"A_2111_KCL01_I2"	I 144.3	BOOL	// SCREW OFF
"A_2111_KCL01_I3"	I 144.4	BOOL	// DRIVE FORWARD SLOWLY
"A_2111_KCL01_I4"	I 144.5	BOOL	// DRIVE BACKWARD SLOWLY
"A_2115_KCL01_I1"	I 160.0	BOOL	// BACKWALL LIFTING
"A_2115_KCL01_I2"	I 160.1	BOOL	// BACKWALL LOWERING
"A_2115_KCL01_I3"	I 160.2	BOOL	// UNCOUPLE
"A_2115_KCL01_I4"	I 160.3	BOOL	// COUPLE
"A_2115_KCL01_I5"	I 160.4	BOOL	// WALL LOCKING
"A_2115_KCL01_I6"	I 160.5	BOOL	// WALL UNLOCKING
"A_2115_KCL01_I7"	I 160.6	BOOL	// HORIZONTAL SCREW ON
"A_2115_KCL01_I8"	I 160.7	BOOL	// DIAGONAL SCREW ON
"A_2115_KCL01_I9"	I 161.0	BOOL	// SCREW STOP
"A_2115_BSA12_I1"	I 161.2	BOOL	// ZERO SPEED MONITOR HORIZONTAL SCREW
"A_2115_BSA17_I1"	I 161.3	BOOL	// ZERO SPEED MONITOR LIFTING SCREW
"A_21_K838R1_I1"	I 162.0	BOOL	// FUSE SWITCH OFF +M212
"A_2199_SHE04_I1"	I 162.1	BOOL	// EMERGENCY-STOP 1 MACHINE DBFL
"A_2199_SHE05_I1"	I 162.2	BOOL	// EMERGENCY-STOP 2 MACHINE DBFL
"A_2199_SHE08_I1"	I 162.3	BOOL	// EMERGENCY-STOP 3 MACHINE DBFL
"A_2115_QYS18_I1"	I 162.4	BOOL	// CLEANING FLAP 1
"A_2115_QYS19_I1"	I 162.5	BOOL	// CLEANING FLAP 2
"A_2115_BTT11_I1"	I 162.6	BOOL	// THERMISTOR HORIZONTAL SCREW
"A_2115_BTT15_I1"	I 162.7	BOOL	// THERMISTOR LIFTING SCREW
"A_2115_BZS42_I1"	I 163.0	BOOL	// COUPLING DRIVE UNLOCKED
"A_2115_BZS43_I1"	I 163.1	BOOL	// COUPLING DRIVE LOCKED
"A_2115_BZS46_I1"	I 163.2	BOOL	// COUPLING DRIVE UNLOCKED
"A_2115_BZS47_I1"	I 163.3	BOOL	// COUPLING DRIVE LOCKED
"A_2150_MXZ01_I1"	I 164.0	BOOL	// AIR-FLAP 1 OPEN
"A_2150_MXZ01_I2"	I 164.1	BOOL	// AIR-FLAP 1 CLOSE
"A_2150_BZS01_I1"	I 164.2	BOOL	// AIR-FLAP 1 CLOSED
"A_2150_BZS02_I1"	I 164.3	BOOL	// AIR-FLAP 1 OPENED
"A_2151_MXZ01_I1"	I 164.4	BOOL	// AIR-FLAP 2 OPEN
"A_2151_MXZ01_I2"	I 164.5	BOOL	// AIR-FLAP 2 CLOSE
"A_2151_BZS01_I1"	I 164.6	BOOL	// AIR-FLAP 2 CLOSED
"A_2151_BZS02_I1"	I 164.7	BOOL	// AIR-FLAP 2 OPENED
"A_2152_MXZ01_I1"	I 165.0	BOOL	// AIR-FLAP 3 OPEN
"A_2152_MXZ01_I2"	I 165.1	BOOL	// AIR-FLAP 3 CLOSE
"A_2152_BZS01_I1"	I 165.2	BOOL	// AIR-FLAP 3 CLOSED
"A_2152_BZS02_I1"	I 165.3	BOOL	// AIR-FLAP 3 OPENED
"A_2154_MXZ01_I1"	I 165.4	BOOL	// WATER PUMP 1
"A_2155_MXZ01_I1"	I 165.5	BOOL	// WATER PUMP 2
"A_2160_MXZ01_I1"	I 165.6	BOOL	// GERM FAN 1
"A_2160_MXZ02_I1"	I 165.7	BOOL	// GERM FAN 2
"A_22_A040Z1_I1"	I 200.0	BOOL	// POWER SUPPLY FAILURE +C22
"A_22_S_H097Z1_I1"	I 200.1	BOOL	// OPERATING ON +C22
"A_22_K091Z1_I1"	I 200.2	BOOL	// FUSE SWITCH OFF +C22
"A_22_A097Z1_I1"	I 200.3	BOOL	// EMERGENCY-STOP +C22
"A_22_A098Z1_I1"	I 200.4	BOOL	// EMERGENCY-STOP +M221/M222
"A_22_Q390Z1_I1"	I 200.5	BOOL	// POWER SUPPLY MACHINE BMKE
"A_22_Q445Z1_I1"	I 200.6	BOOL	// POWER SUPPLY MACHINE DBFL
"A_22_D1B065_I1"	I 200.7	BOOL	// CONTROL 24VDC LIMIT SWITCHES WAY
"A_2299_SHE01_I1"	I 201.0	BOOL	// EMERGENCY-OFF CUSTOMER
"A_2299_SHE02_I1"	I 201.1	BOOL	// EMERGENCY-OFF CUSTOMER
"A_22_A700Z1_I1"	I 201.4	BOOL	// POWER CIRCUIT CABLE CHAIN
"A_22_A106Z1_I1"	I 201.5	BOOL	// EMERGENCY-STOP FROM +C21
"A_22_A800Z1_I1"	I 201.6	BOOL	// POWER CIRCUIT CABLE CHAIN
"A_2201_MXZ01_I1"	I 202.0	BOOL	// BELT CONVEYOR
"A_2202_YMXZ01_I1"	I 202.1	BOOL	// CHUTE DRIVE LEFT SIDE
"A_2202_YMXZ01_I2"	I 202.2	BOOL	// CHUTE DRIVE RIGHT SIDE
"A_2211_MXZ41_I1"	I 203.0	BOOL	// TRAVELING DRIVE
"A_2211_MXZ61_I1"	I 203.2	BOOL	// TURNING SCREW DRIVE 1
"A_2211_MXZ62_I1"	I 203.3	BOOL	// TURNING SCREW DRIVE 2
"A_2211_MXZ63_I1"	I 203.4	BOOL	// TURNING SCREW DRIVE 3
"A_2211_MXZ64_I1"	I 203.5	BOOL	// TURNING SCREW DRIVE 4
"A_2211_MXZ65_I1"	I 203.6	BOOL	// TURNING SCREW DRIVE 5
"A_2211_MXZ66_I1"	I 203.7	BOOL	// TURNING SCREW DRIVE 6
"A_2211_MXZ67_I1"	I 204.0	BOOL	// TURNING SCREW DRIVE 7
"A_2211_MXZ68_I1"	I 204.1	BOOL	// TURNING SCREW DRIVE 8
"A_2211_MXZ69_I1"	I 204.2	BOOL	// TURNING SCREW DRIVE 9
"A_2211_MXZ70_I1"	I 204.3	BOOL	// TURNING SCREW DRIVE 10
"A_2211_MXZ71_I1"	I 204.4	BOOL	// TURNING SCREW DRIVE 11
"A_2211_MXZ72_I1"	I 204.5	BOOL	// TURNING SCREW DRIVE 12
"A_2211_MXZ73_I1"	I 204.6	BOOL	// TURNING SCREW DRIVE 13
"A_2201_SHE20_I1"	I 205.0	BOOL	// CABLE PULL SWITCH RIGHT 1
"A_2201_SHE21_I1"	I 205.1	BOOL	// CABLE PULL SWITCH RIGHT 2
"A_2201_SHE22_I1"	I 205.2	BOOL	// CABLE PULL SWITCH LEFT 1
"A_2201_SHE23_I1"	I 205.3	BOOL	// CABLE PULL SWITCH LEFT 2
"A_2202_QYS21_I1"	I 205.5	BOOL	// DISCHARGE CHUTE LEFT SIDE
"A_2202_QYS22_I1"	I 205.6	BOOL	// DISCHARGE CHUTE RIGHT SIDE
"A_2215_MXZ11_I1"	I 208.0	BOOL	// HORIZONTAL SCREW
"A_2215_MXZ15_I1"	I 208.2	BOOL	// LIFTING SCREW
"A_2215_MXZ21_I1"	I 208.3	BOOL	// LIFTING DEVICE DOWN
"A_2215_MXZ21_I2"	I 208.4	BOOL	// LIFTING DEVICE UP
"A_22_A458Z1_I1"	I 210.0	BOOL	// CLEANING FLAP 1/2
"A_2215_BZS22_I1"	I 210.6	BOOL	// LIFTING DEVICE DOWN
"A_2215_BZS23_I1"	I 210.7	BOOL	// LIFTING DEVICE END POSITION TOP
"A_2245_QXV21_I1"	I 216.0	BOOL	// RUNNING COOLING UNIT GERMINATING
"A_2245_QXV31_I1"	I 216.1	BOOL	// RUNNING COOLING UNIT GERMINATING
"A_2216_BZS12_I1"	I 216.4	BOOL	// SPRINKING WATER LINE OPENED
"A_2216_BZS11_I1"	I 216.5	BOOL	// SPRINKING WATER LINE CLOSED
"A_2231_BZS12_I1"	I 217.2	BOOL	// VALVE HUMIDIFICATION OPENED
"A_2231_BZS11_I1"	I 217.3	BOOL	// VALVE HUMIDIFICATION CLOSED
"A_2201_BSA13_I1"	I 217.4	BOOL	// SPEED CONTROL
"A_2201_BZS14_15_I1"	I 217.6	BOOL	// BELT MONITOR RIGHT
"A_2201_BZS16_17_I1"	I 217.7	BOOL	// BELT MONITOR LEFT
"A_2202_BZS13_I1"	I 218.2	BOOL	// DISCHARGE CHUTE PARKING POSITION
"A_2202_BZS14_I1"	I 218.3	BOOL	// DISCHARGE CHUTE LEFT SIDE
"A_2202_BZS15_I1"	I 218.4	BOOL	// DISCHARGE CHUTE RIGHT SIDE
"A_2212_BZS12_I1"	I 240.0	BOOL	// SPRINKING WATER LINE 1 OPENED
"A_2212_BZS11_I1"	I 240.1	BOOL	// SPRINKING WATER LINE 1 CLOSED
"A_2212_BZS22_I1"	I 240.2	BOOL	// SPRINKING WATER LINE 2 OPENED
"A_2212_BZS21_I1"	I 240.3	BOOL	// SPRINKING WATER LINE 2 CLOSED
"A_2211_KCL01_I1"	I 240.4	BOOL	// SCREW ON
"A_2211_KCL01_I2"	I 240.5	BOOL	// SCREW OFF
"A_2211_KCL01_I3"	I 240.6	BOOL	// DRIVE FORWARD SLOWLY
"A_2211_KCL01_I4"	I 240.7	BOOL	// DRIVE BACKWARD SLOWLY
"A_2211_KCL01_I5"	I 241.0	BOOL	// DRIVE FORWARD FASTER
"A_2211_KCL01_I6"	I 241.1	BOOL	// DRIVE BACKWARD FASTER
"A_2211_BZS44_I1"	I 241.2	BOOL	// TRAVELING DRIVE STOP LEFT SIDE
"A_2211_BZS46_I1"	I 241.3	BOOL	// TRAVELING DRIVE STOP RIGHT SIDE
"A_22_K738R1_I1"	I 242.0	BOOL	// FUSE SWITCH OFF +M221
"A_22_A408Z1_I1"	I 242.1	BOOL	// BUMPER SWITCHED-OFF
"A_2299_SHE03_I1"	I 242.2	BOOL	// EMERGENCY-STOP 1 MACHINE BMKE
"A_2299_SHE06_I1"	I 242.3	BOOL	// EMERGENCY-STOP 2 MACHINE BMKE
"A_2211_QYS43_I1"	I 242.4	BOOL	// TRAVELING DRIVE SAFETY STLEFT SIDE
"A_2211_QYS45_I1"	I 242.5	BOOL	// TRAVELING DRIVE SAFETY STRIGHT SIDE
"A_2299_SHE20_I1"	I 242.6	BOOL	// CABLE PULL SWITCH RIGHT
"A_2299_SHE21_I1"	I 242.7	BOOL	// CABLE PULL SWITCH LEFT
"A_2211_BZS22_I1"	I 243.0	BOOL	// COUPLING DRIVE UNLOCKED
"A_2211_BZS23_I1"	I 243.1	BOOL	// COUPLING DRIVE LOCKED
"A_2211_BZS26_I1"	I 243.2	BOOL	// COUPLING DRIVE UNLOCKED
"A_2211_BZS27_I1"	I 243.3	BOOL	// COUPLING DRIVE LOCKED
"A_2211_BZS32_I1"	I 243.4	BOOL	// COUPLING DRIVE UNLOCKED
"A_2211_BZS33_I1"	I 243.5	BOOL	// COUPLING DRIVE LOCKED
"A_2211_BZS36_I1"	I 243.6	BOOL	// COUPLING DRIVE UNLOCKED
"A_2211_BZS37_I1"	I 243.7	BOOL	// COUPLING DRIVE LOCKED
"A_2215_KCL01_I1"	I 260.0	BOOL	// BACKWALL LIFTING
"A_2215_KCL01_I2"	I 260.1	BOOL	// BACKWALL LOWERING
"A_2215_KCL01_I3"	I 260.2	BOOL	// UNCOUPLE
"A_2215_KCL01_I4"	I 260.3	BOOL	// COUPLE
"A_2215_KCL01_I5"	I 260.4	BOOL	// WALL LOCKING
"A_2215_KCL01_I6"	I 260.5	BOOL	// WALL UNLOCKING
"A_2215_KCL01_I7"	I 260.6	BOOL	// HORIZONTAL SCREW ON
"A_2215_KCL01_I8"	I 260.7	BOOL	// DIAGONAL SCREW ON
"A_2215_KCL01_I9"	I 261.0	BOOL	// SCREW STOP
"A_2215_BSA12_I1"	I 261.2	BOOL	// ZERO SPEED MONITOR HORIZONTAL SCREW
"A_2215_BSA17_I1"	I 261.3	BOOL	// ZERO SPEED MONITOR LIFTING SCREW
"A_22_K838R1_I1"	I 262.0	BOOL	// FUSE SWITCH OFF +M222
"A_2299_SHE04_I1"	I 262.1	BOOL	// EMERGENCY-STOP 1 MACHINE DBFL
"A_2299_SHE05_I1"	I 262.2	BOOL	// EMERGENCY-STOP 2 MACHINE DBFL
"A_2299_SHE08_I1"	I 262.3	BOOL	// EMERGENCY-STOP 3 MACHINE DBFL
"A_2215_QYS18_I1"	I 262.4	BOOL	// CLEANING FLAP 1
"A_2215_QYS19_I1"	I 262.5	BOOL	// CLEANING FLAP 2
"A_2215_BTT11_I1"	I 262.6	BOOL	// THERMISTOR HORIZONTAL SCREW
"A_2215_BTT15_I1"	I 262.7	BOOL	// THERMISTOR LIFTING SCREW
"A_2215_BZS42_I1"	I 263.0	BOOL	// COUPLING DRIVE UNLOCKED
"A_2215_BZS43_I1"	I 263.1	BOOL	// COUPLING DRIVE LOCKED
"A_2215_BZS46_I1"	I 263.2	BOOL	// COUPLING DRIVE UNLOCKED
"A_2215_BZS47_I1"	I 263.3	BOOL	// COUPLING DRIVE LOCKED
"A_2250_MXZ01_I1"	I 264.0	BOOL	// AIR-FLAP 1 OPEN
"A_2250_MXZ01_I2"	I 264.1	BOOL	// AIR-FLAP 1 CLOSE
"A_2250_BZS01_I1"	I 264.2	BOOL	// AIR-FLAP 1 CLOSED
"A_2250_BZS02_I1"	I 264.3	BOOL	// AIR-FLAP 1 OPENED
"A_2251_MXZ01_I1"	I 264.4	BOOL	// AIR-FLAP 2 OPEN
"A_2251_MXZ01_I2"	I 264.5	BOOL	// AIR-FLAP 2 CLOSE
"A_2251_BZS01_I1"	I 264.6	BOOL	// AIR-FLAP 2 CLOSED
"A_2251_BZS02_I1"	I 264.7	BOOL	// AIR-FLAP 2 OPENED
"A_2252_MXZ01_I1"	I 265.0	BOOL	// AIR-FLAP 3 OPEN
"A_2252_MXZ01_I2"	I 265.1	BOOL	// AIR-FLAP 3 CLOSE
"A_2252_BZS01_I1"	I 265.2	BOOL	// AIR-FLAP 3 CLOSED
"A_2252_BZS02_I1"	I 265.3	BOOL	// AIR-FLAP 3 OPENED
"A_2254_MXZ01_I1"	I 265.4	BOOL	// WATER PUMP 1
"A_2255_MXZ01_I1"	I 265.5	BOOL	// WATER PUMP 2
"A_2260_MXZ01_I1"	I 265.6	BOOL	// GERM FAN 1
"A_2260_MXZ02_I1"	I 265.7	BOOL	// GERM FAN 2
"A_23_A040Z1_I1"	I 300.0	BOOL	// POWER SUPPLY FAILURE +C23
"A_23_S_H097Z1_I1"	I 300.1	BOOL	// OPERATING ON +C23
"A_23_K091Z1_I1"	I 300.2	BOOL	// FUSE SWITCH OFF +C23
"A_23_A097Z1_I1"	I 300.3	BOOL	// EMERGENCY-STOP +C23
"A_23_A098Z1_I1"	I 300.4	BOOL	// EMERGENCY-STOP +M231/M232
"A_23_Q390Z1_I1"	I 300.5	BOOL	// POWER SUPPLY MACHINE BMKE
"A_23_Q445Z1_I1"	I 300.6	BOOL	// POWER SUPPLY MACHINE DBFL
"A_23_D1B065_I1"	I 300.7	BOOL	// CONTROL 24VDC LIMIT SWITCHES WAY
"A_2399_SHE01_I1"	I 301.0	BOOL	// EMERGENCY-OFF CUSTOMER
"A_2399_SHE02_I1"	I 301.1	BOOL	// EMERGENCY-OFF CUSTOMER
"A_23_A700Z1_I1"	I 301.4	BOOL	// POWER CIRCUIT CABLE CHAIN
"A_23_A106Z1_I1"	I 301.5	BOOL	// EMERGENCY-STOP FROM +C24
"A_23_A800Z1_I1"	I 301.6	BOOL	// POWER CIRCUIT CABLE CHAIN
"A_2301_MXZ01_I1"	I 302.0	BOOL	// BELT CONVEYOR
"A_2302_YMXZ01_I1"	I 302.1	BOOL	// CHUTE DRIVE LEFT SIDE
"A_2302_YMXZ01_I2"	I 302.2	BOOL	// CHUTE DRIVE RIGHT SIDE
"A_2311_MXZ41_I1"	I 303.0	BOOL	// TRAVELING DRIVE
"A_2311_MXZ61_I1"	I 303.2	BOOL	// TURNING SCREW DRIVE 1
"A_2311_MXZ62_I1"	I 303.3	BOOL	// TURNING SCREW DRIVE 2
"A_2311_MXZ63_I1"	I 303.4	BOOL	// TURNING SCREW DRIVE 3
"A_2311_MXZ64_I1"	I 303.5	BOOL	// TURNING SCREW DRIVE 4
"A_2311_MXZ65_I1"	I 303.6	BOOL	// TURNING SCREW DRIVE 5
"A_2311_MXZ66_I1"	I 303.7	BOOL	// TURNING SCREW DRIVE 6
"A_2311_MXZ67_I1"	I 304.0	BOOL	// TURNING SCREW DRIVE 7
"A_2311_MXZ68_I1"	I 304.1	BOOL	// TURNING SCREW DRIVE 8
"A_2311_MXZ69_I1"	I 304.2	BOOL	// TURNING SCREW DRIVE 9
"A_2311_MXZ70_I1"	I 304.3	BOOL	// TURNING SCREW DRIVE 10
"A_2311_MXZ71_I1"	I 304.4	BOOL	// TURNING SCREW DRIVE 12
"A_2311_MXZ72_I1"	I 304.5	BOOL	// TURNING SCREW DRIVE 12
"A_2311_MXZ73_I1"	I 304.6	BOOL	// TURNING SCREW DRIVE 13
"A_2301_SHE20_I1"	I 305.0	BOOL	// CABLE PULL SWITCH RIGHT 1
"A_2301_SHE21_I1"	I 305.1	BOOL	// CABLE PULL SWITCH RIGHT 2
"A_2301_SHE22_I1"	I 305.2	BOOL	// CABLE PULL SWITCH LEFT 1
"A_2301_SHE23_I1"	I 305.3	BOOL	// CABLE PULL SWITCH LEFT 2
"A_2302_QYS21_I1"	I 305.5	BOOL	// DISCHARGE CHUTE LEFT SIDE
"A_2302_QYS22_I1"	I 305.6	BOOL	// DISCHARGE CHUTE RIGHT SIDE
"A_2315_MXZ11_I1"	I 308.0	BOOL	// HORIZONTAL SCREW
"A_2315_MXZ15_I1"	I 308.2	BOOL	// LIFTING SCREW
"A_2315_MXZ21_I1"	I 308.3	BOOL	// LIFTING DEVICE DOWN
"A_2315_MXZ21_I2"	I 308.4	BOOL	// LIFTING DEVICE UP
"A_23_A458Z1_I1"	I 310.0	BOOL	// CLEANING FLAP 1/2
"A_2315_BZS22_I1"	I 310.6	BOOL	// LIFTING DEVICE DOWN
"A_2315_BZS23_I1"	I 310.7	BOOL	// LIFTING DEVICE END POSITION TOP
"A_2345_QXV21_I1"	I 316.0	BOOL	// RUNNING COOLING UNIT GERMINATING
"A_2345_QXV31_I1"	I 316.1	BOOL	// RUNNING COOLING UNIT GERMINATING
"A_2316_BZS12_I1"	I 316.4	BOOL	// SPRINKING WATER LINE OPENED
"A_2316_BZS11_I1"	I 316.5	BOOL	// SPRINKING WATER LINE CLOSED
"A_2331_BZS12_I1"	I 317.2	BOOL	// VALVE HUMIDIFICATION OPENED
"A_2331_BZS11_I1"	I 317.3	BOOL	// VALVE HUMIDIFICATION CLOSED
"A_2301_BSA13_I1"	I 317.4	BOOL	// SPEED CONTROL
"A_2301_BZS14_15_I1"	I 317.6	BOOL	// BELT MONITOR RIGHT
"A_2301_BZS16_17_I1"	I 317.7	BOOL	// BELT MONITOR LEFT
"A_2302_BZS13_I1"	I 318.2	BOOL	// DISCHARGE CHUTE PARKING POSITION
"A_2302_BZS14_I1"	I 318.3	BOOL	// DISCHARGE CHUTE LEFT SIDE
"A_2302_BZS15_I1"	I 318.4	BOOL	// DISCHARGE CHUTE RIGHT SIDE
"A_2312_BZS12_I1"	I 340.0	BOOL	// SPRINKING WATER LINE 1 OPENED
"A_2312_BZS11_I1"	I 340.1	BOOL	// SPRINKING WATER LINE 1 CLOSED
"A_2312_BZS22_I1"	I 340.2	BOOL	// SPRINKING WATER LINE 2 OPENED
"A_2312_BZS21_I1"	I 340.3	BOOL	// SPRINKING WATER LINE 2 CLOSED
"A_2311_KCL01_I1"	I 340.4	BOOL	// SCREW ON
"A_2311_KCL01_I2"	I 340.5	BOOL	// SCREW OFF
"A_2311_KCL01_I3"	I 340.6	BOOL	// DRIVE FORWARD SLOWLY
"A_2311_KCL01_I4"	I 340.7	BOOL	// DRIVE BACKWARD SLOWLY
"A_2311_KCL01_I5"	I 341.0	BOOL	// DRIVE FORWARD FASTER
"A_2311_KCL01_I6"	I 341.1	BOOL	// DRIVE BACKWARD FASTER
"A_2311_BZS44_I1"	I 341.2	BOOL	// TRAVELING DRIVE STOP LEFT SIDE
"A_2311_BZS46_I1"	I 341.3	BOOL	// TRAVELING DRIVE STOP RIGHT SIDE
"A_23_K738R1_I1"	I 342.0	BOOL	// FUSE SWITCH OFF +M231
"A_23_A408Z1_I1"	I 342.1	BOOL	// BUMPER SWITCHED-OFF
"A_2399_SHE03_I1"	I 342.2	BOOL	// EMERGENCY-STOP 1 MACHINE BMKE
"A_2399_SHE06_I1"	I 342.3	BOOL	// EMERGENCY-STOP 2 MACHINE BMKE
"A_2311_QYS43_I1"	I 342.4	BOOL	// TRAVELING DRIVE SAFETY STLEFT SIDE
"A_2311_QYS45_I1"	I 342.5	BOOL	// TRAVELING DRIVE SAFETY STRIGHT SIDE
"A_2399_SHE20_I1"	I 342.6	BOOL	// CABLE PULL SWITCH RIGHT
"A_2399_SHE21_I1"	I 342.7	BOOL	// CABLE PULL SWITCH LEFT
"A_2311_BZS22_I1"	I 343.0	BOOL	// COUPLING DRIVE UNLOCKED
"A_2311_BZS23_I1"	I 343.1	BOOL	// COUPLING DRIVE LOCKED
"A_2311_BZS26_I1"	I 343.2	BOOL	// COUPLING DRIVE UNLOCKED
"A_2311_BZS27_I1"	I 343.3	BOOL	// COUPLING DRIVE LOCKED
"A_2311_BZS32_I1"	I 343.4	BOOL	// COUPLING DRIVE UNLOCKED
"A_2311_BZS33_I1"	I 343.5	BOOL	// COUPLING DRIVE LOCKED
"A_2311_BZS36_I1"	I 343.6	BOOL	// COUPLING DRIVE UNLOCKED
"A_2311_BZS37_I1"	I 343.7	BOOL	// COUPLING DRIVE LOCKED
"A_2315_KCL01_I1"	I 360.0	BOOL	// BACKWALL LIFTING
"A_2315_KCL01_I2"	I 360.1	BOOL	// BACKWALL LOWERING
"A_2315_KCL01_I3"	I 360.2	BOOL	// UNCOUPLE
"A_2315_KCL01_I4"	I 360.3	BOOL	// COUPLE
"A_2315_KCL01_I5"	I 360.4	BOOL	// WALL LOCKING
"A_2315_KCL01_I6"	I 360.5	BOOL	// WALL UNLOCKING
"A_2315_KCL01_I7"	I 360.6	BOOL	// HORIZONTAL SCREW ON
"A_2315_KCL01_I8"	I 360.7	BOOL	// DIAGONAL SCREW ON
"A_2315_KCL01_I9"	I 361.0	BOOL	// SCREW STOP
"A_2315_BSA12_I1"	I 361.2	BOOL	// ZERO SPEED MONITOR HORIZONTAL SCREW
"A_2315_BSA17_I1"	I 361.3	BOOL	// ZERO SPEED MONITOR LIFTING SCREW
"A_23_K838R1_I1"	I 362.0	BOOL	// FUSE SWITCH OFF +M232
"A_2399_SHE04_I1"	I 362.1	BOOL	// EMERGENCY-STOP 1 MACHINE DBFL
"A_2399_SHE05_I1"	I 362.2	BOOL	// EMERGENCY-STOP 2 MACHINE DBFL
"A_2399_SHE08_I1"	I 362.3	BOOL	// EMERGENCY-STOP 3 MACHINE DBFL
"A_2315_QYS18_I1"	I 362.4	BOOL	// CLEANING FLAP 1
"A_2315_QYS19_I1"	I 362.5	BOOL	// CLEANING FLAP 2
"A_2315_BTT11_I1"	I 362.6	BOOL	// THERMISTOR HORIZONTAL SCREW
"A_2315_BTT15_I1"	I 362.7	BOOL	// THERMISTOR LIFTING SCREW
"A_2315_BZS42_I1"	I 363.0	BOOL	// COUPLING DRIVE UNLOCKED
"A_2315_BZS43_I1"	I 363.1	BOOL	// COUPLING DRIVE LOCKED
"A_2315_BZS46_I1"	I 363.2	BOOL	// COUPLING DRIVE UNLOCKED
"A_2315_BZS47_I1"	I 363.3	BOOL	// COUPLING DRIVE LOCKED
"A_2350_MXZ01_I1"	I 364.0	BOOL	// AIR-FLAP 1 OPEN
"A_2350_MXZ01_I2"	I 364.1	BOOL	// AIR-FLAP 1 CLOSE
"A_2350_BZS01_I1"	I 364.2	BOOL	// AIR-FLAP 1 CLOSED
"A_2350_BZS02_I1"	I 364.3	BOOL	// AIR-FLAP 1 OPENED
"A_2351_MXZ01_I1"	I 364.4	BOOL	// AIR-FLAP 2 OPEN
"A_2351_MXZ01_I2"	I 364.5	BOOL	// AIR-FLAP 2 CLOSE
"A_2351_BZS01_I1"	I 364.6	BOOL	// AIR-FLAP 2 CLOSED
"A_2351_BZS02_I1"	I 364.7	BOOL	// AIR-FLAP 2 OPENED
"A_2352_MXZ01_I1"	I 365.0	BOOL	// AIR-FLAP 3 OPEN
"A_2352_MXZ01_I2"	I 365.1	BOOL	// AIR-FLAP 3 CLOSE
"A_2352_BZS01_I1"	I 365.2	BOOL	// AIR-FLAP 3 CLOSED
"A_2352_BZS02_I1"	I 365.3	BOOL	// AIR-FLAP 3 OPENED
"A_2354_MXZ01_I1"	I 365.4	BOOL	// WATER PUMP 1
"A_2355_MXZ01_I1"	I 365.5	BOOL	// WATER PUMP 2
"A_2360_MXZ01_I1"	I 365.6	BOOL	// GERM FAN 1
"A_2360_MXZ02_I1"	I 365.7	BOOL	// GERM FAN 2
"A_24_A040Z1_I1"	I 400.0	BOOL	// POWER SUPPLY FAILURE +C24
"A_24_S_H097Z1_I1"	I 400.1	BOOL	// OPERATING ON +C24
"A_24_K091Z1_I1"	I 400.2	BOOL	// FUSE SWITCH OFF +C24
"A_24_A097Z1_I1"	I 400.3	BOOL	// EMERGENCY-STOP +C24
"A_24_A098Z1_I1"	I 400.4	BOOL	// EMERGENCY-STOP +M241/M242
"A_24_Q390Z1_I1"	I 400.5	BOOL	// POWER SUPPLY MACHINE BMKE
"A_24_Q445Z1_I1"	I 400.6	BOOL	// POWER SUPPLY MACHINE DBFL
"A_24_D1B065_I1"	I 400.7	BOOL	// CONTROL 24VDC LIMIT SWITCHES WAY
"A_2499_SHE01_I1"	I 401.0	BOOL	// EMERGENCY-OFF CUSTOMER
"A_2499_SHE02_I1"	I 401.1	BOOL	// EMERGENCY-OFF CUSTOMER
"A_24_A700Z1_I1"	I 401.4	BOOL	// POWER CIRCUIT CABLE CHAIN
"A_24_A106Z1_I1"	I 401.5	BOOL	// EMERGENCY-STOP FROM +C23
"A_24_A800Z1_I1"	I 401.6	BOOL	// POWER CIRCUIT CABLE CHAIN
"A_2401_MXZ01_I1"	I 402.0	BOOL	// BELT CONVEYOR
"A_2402_YMXZ01_I1"	I 402.1	BOOL	// CHUTE DRIVE LEFT SIDE
"A_2402_YMXZ01_I2"	I 402.2	BOOL	// CHUTE DRIVE RIGHT SIDE
"A_2411_MXZ41_I1"	I 403.0	BOOL	// TRAVELING DRIVE
"A_2411_MXZ61_I1"	I 403.2	BOOL	// TURNING SCREW DRIVE 1
"A_2411_MXZ62_I1"	I 403.3	BOOL	// TURNING SCREW DRIVE 2
"A_2411_MXZ63_I1"	I 403.4	BOOL	// TURNING SCREW DRIVE 3
"A_2411_MXZ64_I1"	I 403.5	BOOL	// TURNING SCREW DRIVE 4
"A_2411_MXZ65_I1"	I 403.6	BOOL	// TURNING SCREW DRIVE 5
"A_2411_MXZ66_I1"	I 403.7	BOOL	// TURNING SCREW DRIVE 6
"A_2411_MXZ67_I1"	I 404.0	BOOL	// TURNING SCREW DRIVE 7
"A_2411_MXZ68_I1"	I 404.1	BOOL	// TURNING SCREW DRIVE 8
"A_2411_MXZ69_I1"	I 404.2	BOOL	// TURNING SCREW DRIVE 9
"A_2411_MXZ70_I1"	I 404.3	BOOL	// TURNING SCREW DRIVE 10
"A_2411_MXZ71_I1"	I 404.4	BOOL	// TURNING SCREW DRIVE 11
"A_2411_MXZ72_I1"	I 404.5	BOOL	// TURNING SCREW DRIVE 12
"A_2411_MXZ73_I1"	I 404.6	BOOL	// TURNING SCREW DRIVE 13
"A_2401_SHE20_I1"	I 405.0	BOOL	// CABLE PULL SWITCH RIGHT 1
"A_2401_SHE21_I1"	I 405.1	BOOL	// CABLE PULL SWITCH RIGHT 2
"A_2401_SHE22_I1"	I 405.2	BOOL	// CABLE PULL SWITCH LEFT 1
"A_2401_SHE23_I1"	I 405.3	BOOL	// CABLE PULL SWITCH LEFT 2
"A_2402_QYS21_I1"	I 405.5	BOOL	// DISCHARGE CHUTE LEFT SIDE
"A_2402_QYS22_I1"	I 405.6	BOOL	// DISCHARGE CHUTE RIGHT SIDE
"A_2415_MXZ11_I1"	I 408.0	BOOL	// HORIZONTAL SCREW
"A_2415_MXZ15_I1"	I 408.2	BOOL	// LIFTING SCREW
"A_2415_MXZ21_I1"	I 408.3	BOOL	// LIFTING DEVICE DOWN
"A_2415_MXZ21_I2"	I 408.4	BOOL	// LIFTING DEVICE UP
"A_24_A458Z1_I1"	I 410.0	BOOL	// CLEANING FLAP 1/2
"A_2415_BZS22_I1"	I 410.6	BOOL	// LIFTING DEVICE DOWN
"A_2415_BZS23_I1"	I 410.7	BOOL	// LIFTING DEVICE END POSITION TOP
"A_2445_QXV21_I1"	I 416.0	BOOL	// RUNNING COOLING UNIT GERMINATING
"A_2445_QXV31_I1"	I 416.1	BOOL	// RUNNING COOLING UNIT GERMINATING
"A_2416_BZS12_I1"	I 416.4	BOOL	// SPRINKING WATER LINE OPENED
"A_2416_BZS11_I1"	I 416.5	BOOL	// SPRINKING WATER LINE CLOSED
"A_2431_BZS12_I1"	I 417.2	BOOL	// VALVE HUMIDIFICATION OPENED
"A_2431_BZS11_I1"	I 417.3	BOOL	// VALVE HUMIDIFICATION CLOSED
"A_2401_BSA13_I1"	I 417.4	BOOL	// SPEED CONTROL
"A_2401_BZS14_15_I1"	I 417.6	BOOL	// BELT MONITOR RIGHT
"A_2401_BZS16_17_I1"	I 417.7	BOOL	// BELT MONITOR LEFT
"A_2402_BZS13_I1"	I 418.2	BOOL	// DISCHARGE CHUTE PARKING POSITION
"A_2402_BZS14_I1"	I 418.3	BOOL	// DISCHARGE CHUTE LEFT SIDE
"A_2402_BZS15_I1"	I 418.4	BOOL	// DISCHARGE CHUTE RIGHT SIDE
"A_2412_BZS12_I1"	I 440.0	BOOL	// SPRINKING WATER LINE 1 OPENED
"A_2412_BZS11_I1"	I 440.1	BOOL	// SPRINKING WATER LINE 1 CLOSED
"A_2412_BZS22_I1"	I 440.2	BOOL	// SPRINKING WATER LINE 2 OPENED
"A_2412_BZS21_I1"	I 440.3	BOOL	// SPRINKING WATER LINE 2 CLOSED
"A_2411_KCL01_I1"	I 440.4	BOOL	// SCREW ON
"A_2411_KCL01_I2"	I 440.5	BOOL	// SCREW OFF
"A_2411_KCL01_I3"	I 440.6	BOOL	// DRIVE FORWARD SLOWLY
"A_2411_KCL01_I4"	I 440.7	BOOL	// DRIVE BACKWARD SLOWLY
"A_2411_KCL01_I5"	I 441.0	BOOL	// DRIVE FORWARD FASTER
"A_2411_KCL01_I6"	I 441.1	BOOL	// DRIVE BACKWARD FASTER
"A_2411_BZS44_I1"	I 441.2	BOOL	// TRAVELING DRIVE STOP LEFT SIDE
"A_2411_BZS46_I1"	I 441.3	BOOL	// TRAVELING DRIVE STOP RIGHT SIDE
"A_24_K738R1_I1"	I 442.0	BOOL	// FUSE SWITCH OFF +M241
"A_24_A408Z1_I1"	I 442.1	BOOL	// BUMPER SWITCHED-OFF
"A_2499_SHE03_I1"	I 442.2	BOOL	// EMERGENCY-STOP 1 MACHINE BMKE
"A_2499_SHE06_I1"	I 442.3	BOOL	// EMERGENCY-STOP 2 MACHINE BMKE
"A_2411_QYS43_I1"	I 442.4	BOOL	// TRAVELING DRIVE SAFETY STLEFT SIDE
"A_2411_QYS45_I1"	I 442.5	BOOL	// TRAVELING DRIVE SAFETY STRIGHT SIDE
"A_2499_SHE20_I1"	I 442.6	BOOL	// CABLE PULL SWITCH RIGHT
"A_2499_SHE21_I1"	I 442.7	BOOL	// CABLE PULL SWITCH LEFT
"A_2411_BZS22_I1"	I 443.0	BOOL	// COUPLING DRIVE UNLOCKED
"A_2411_BZS23_I1"	I 443.1	BOOL	// COUPLING DRIVE LOCKED
"A_2411_BZS26_I1"	I 443.2	BOOL	// COUPLING DRIVE UNLOCKED
"A_2411_BZS27_I1"	I 443.3	BOOL	// COUPLING DRIVE LOCKED
"A_2411_BZS32_I1"	I 443.4	BOOL	// COUPLING DRIVE UNLOCKED
"A_2411_BZS33_I1"	I 443.5	BOOL	// COUPLING DRIVE LOCKED
"A_2411_BZS36_I1"	I 443.6	BOOL	// COUPLING DRIVE UNLOCKED
"A_2411_BZS37_I1"	I 443.7	BOOL	// COUPLING DRIVE LOCKED
"A_2415_KCL01_I1"	I 460.0	BOOL	// BACKWALL LIFTING
"A_2415_KCL01_I2"	I 460.1	BOOL	// BACKWALL LOWERING
"A_2415_KCL01_I3"	I 460.2	BOOL	// UNCOUPLE
"A_2415_KCL01_I4"	I 460.3	BOOL	// COUPLE
"A_2415_KCL01_I5"	I 460.4	BOOL	// WALL LOCKING
"A_2415_KCL01_I6"	I 460.5	BOOL	// WALL UNLOCKING
"A_2415_KCL01_I7"	I 460.6	BOOL	// HORIZONTAL SCREW ON
"A_2415_KCL01_I8"	I 460.7	BOOL	// DIAGONAL SCREW ON
"A_2415_KCL01_I9"	I 461.0	BOOL	// SCREW STOP
"A_2415_BSA12_I1"	I 461.2	BOOL	// ZERO SPEED MONITOR HORIZONTAL SCREW
"A_2415_BSA17_I1"	I 461.3	BOOL	// ZERO SPEED MONITOR LIFTING SCREW
"A_24_K838R1_I1"	I 462.0	BOOL	// FUSE SWITCH OFF +M242
"A_2499_SHE04_I1"	I 462.1	BOOL	// EMERGENCY-STOP 1 MACHINE DBFL
"A_2499_SHE05_I1"	I 462.2	BOOL	// EMERGENCY-STOP 2 MACHINE DBFL
"A_2499_SHE08_I1"	I 462.3	BOOL	// EMERGENCY-STOP 3 MACHINE DBFL
"A_2415_QYS18_I1"	I 462.4	BOOL	// CLEANING FLAP 1
"A_2415_QYS19_I1"	I 462.5	BOOL	// CLEANING FLAP 2
"A_2415_BTT11_I1"	I 462.6	BOOL	// THERMISTOR HORIZONTAL SCREW
"A_2415_BTT15_I1"	I 462.7	BOOL	// THERMISTOR LIFTING SCREW
"A_2415_BZS42_I1"	I 463.0	BOOL	// COUPLING DRIVE UNLOCKED
"A_2415_BZS43_I1"	I 463.1	BOOL	// COUPLING DRIVE LOCKED
"A_2415_BZS46_I1"	I 463.2	BOOL	// COUPLING DRIVE UNLOCKED
"A_2415_BZS47_I1"	I 463.3	BOOL	// COUPLING DRIVE LOCKED
"A_2450_MXZ01_I1"	I 464.0	BOOL	// AIR-FLAP 1 OPEN
"A_2450_MXZ01_I2"	I 464.1	BOOL	// AIR-FLAP 1 CLOSE
"A_2450_BZS01_I1"	I 464.2	BOOL	// AIR-FLAP 1 CLOSED
"A_2450_BZS02_I1"	I 464.3	BOOL	// AIR-FLAP 1 OPENED
"A_2451_MXZ01_I1"	I 464.4	BOOL	// AIR-FLAP 2 OPEN
"A_2451_MXZ01_I2"	I 464.5	BOOL	// AIR-FLAP 2 CLOSE
"A_2451_BZS01_I1"	I 464.6	BOOL	// AIR-FLAP 2 CLOSED
"A_2451_BZS02_I1"	I 464.7	BOOL	// AIR-FLAP 2 OPENED
"A_2452_MXZ01_I1"	I 465.0	BOOL	// AIR-FLAP 3 OPEN
"A_2452_MXZ01_I2"	I 465.1	BOOL	// AIR-FLAP 3 CLOSE
"A_2452_BZS01_I1"	I 465.2	BOOL	// AIR-FLAP 3 CLOSED
"A_2452_BZS02_I1"	I 465.3	BOOL	// AIR-FLAP 3 OPENED
"A_2454_MXZ01_I1"	I 465.4	BOOL	// WATER PUMP 1
"A_2455_MXZ01_I1"	I 465.5	BOOL	// WATER PUMP 2
"A_2460_MXZ01_I1"	I 465.6	BOOL	// GERM FAN 1
"A_2460_MXZ02_I1"	I 465.7	BOOL	// GERM FAN 2
"A_25_A040Z1_I1"	I 500.0	BOOL	// POWER SUPPLY FAILURE +C25
"A_25_S_H097Z1_I1"	I 500.1	BOOL	// OPERATING ON +C25
"A_25_K091Z1_I1"	I 500.2	BOOL	// FUSE SWITCH OFF +C25
"A_25_A097Z1_I1"	I 500.3	BOOL	// EMERGENCY-STOP +C25
"A_25_A098Z1_I1"	I 500.4	BOOL	// EMERGENCY-STOP +M251/M252
"A_25_Q390Z1_I1"	I 500.5	BOOL	// POWER SUPPLY MACHINE BMKE
"A_25_Q445Z1_I1"	I 500.6	BOOL	// POWER SUPPLY MACHINE DBFL
"A_25_D1B065_I1"	I 500.7	BOOL	// CONTROL 24VDC LIMIT SWITCHES WAY
"A_2599_SHE01_I1"	I 501.0	BOOL	// EMERGENCY-OFF CUSTOMER
"A_2599_SHE02_I1"	I 501.1	BOOL	// EMERGENCY-OFF CUSTOMER
"A_25_A700Z1_I1"	I 501.4	BOOL	// POWER CIRCUIT CABLE CHAIN
"A_25_A106Z1_I1"	I 501.5	BOOL	// EMERGENCY-STOP FROM +C26
"A_25_A800Z1_I1"	I 501.6	BOOL	// POWER CIRCUIT CABLE CHAIN
"A_2501_MXZ01_I1"	I 502.0	BOOL	// BELT CONVEYOR
"A_2502_YMXZ01_I1"	I 502.1	BOOL	// CHUTE DRIVE LEFT SIDE
"A_2502_YMXZ01_I2"	I 502.2	BOOL	// CHUTE DRIVE RIGHT SIDE
"A_2511_MXZ41_I1"	I 503.0	BOOL	// TRAVELING DRIVE
"A_2511_MXZ61_I1"	I 503.2	BOOL	// TURNING SCREW DRIVE 1
"A_2511_MXZ62_I1"	I 503.3	BOOL	// TURNING SCREW DRIVE 2
"A_2511_MXZ63_I1"	I 503.4	BOOL	// TURNING SCREW DRIVE 3
"A_2511_MXZ64_I1"	I 503.5	BOOL	// TURNING SCREW DRIVE 4
"A_2511_MXZ65_I1"	I 503.6	BOOL	// TURNING SCREW DRIVE 5
"A_2511_MXZ66_I1"	I 503.7	BOOL	// TURNING SCREW DRIVE 6
"A_2511_MXZ67_I1"	I 504.0	BOOL	// TURNING SCREW DRIVE 7
"A_2511_MXZ68_I1"	I 504.1	BOOL	// TURNING SCREW DRIVE 8
"A_2511_MXZ69_I1"	I 504.2	BOOL	// TURNING SCREW DRIVE 9
"A_2511_MXZ70_I1"	I 504.3	BOOL	// TURNING SCREW DRIVE 10
"A_2511_MXZ71_I1"	I 504.4	BOOL	// TURNING SCREW DRIVE 11
"A_2511_MXZ72_I1"	I 504.5	BOOL	// TURNING SCREW DRIVE 12
"A_2511_MXZ73_I1"	I 504.6	BOOL	// TURNING SCREW DRIVE 13
"A_2501_SHE20_I1"	I 505.0	BOOL	// CABLE PULL SWITCH RIGHT 1
"A_2501_SHE21_I1"	I 505.1	BOOL	// CABLE PULL SWITCH RIGHT 2
"A_2501_SHE22_I1"	I 505.2	BOOL	// CABLE PULL SWITCH LEFT 1
"A_2501_SHE23_I1"	I 505.3	BOOL	// CABLE PULL SWITCH LEFT 2
"A_2502_QYS21_I1"	I 505.5	BOOL	// DISCHARGE CHUTE LEFT SIDE
"A_2502_QYS22_I1"	I 505.6	BOOL	// DISCHARGE CHUTE RIGHT SIDE
"A_2515_MXZ11_I1"	I 508.0	BOOL	// HORIZONTAL SCREW
"A_2515_MXZ15_I1"	I 508.2	BOOL	// LIFTING SCREW
"A_2515_MXZ21_I1"	I 508.3	BOOL	// LIFTING DEVICE DOWN
"A_2515_MXZ21_I2"	I 508.4	BOOL	// LIFTING DEVICE UP
"A_25_A458Z1_I1"	I 510.0	BOOL	// CLEANING FLAP 1/2
"A_2515_BZS22_I1"	I 510.6	BOOL	// LIFTING DEVICE DOWN
"A_2515_BZS23_I1"	I 510.7	BOOL	// LIFTING DEVICE END POSITION TOP
"A_2545_QXV21_I1"	I 516.0	BOOL	// RUNNING COOLING UNIT GERMINATING
"A_2545_QXV31_I1"	I 516.1	BOOL	// RUNNING COOLING UNIT GERMINATING
"A_2516_BZS12_I1"	I 516.4	BOOL	// SPRINKING WATER LINE OPENED
"A_2516_BZS11_I1"	I 516.5	BOOL	// SPRINKING WATER LINE CLOSED
"A_2531_BZS12_I1"	I 517.2	BOOL	// VALVE HUMIDIFICATION OPENED
"A_2531_BZS11_I1"	I 517.3	BOOL	// VALVE HUMIDIFICATION CLOSED
"A_2501_BSA13_I1"	I 517.4	BOOL	// SPEED CONTROL
"A_2501_BZS14_15_I1"	I 517.6	BOOL	// BELT MONITOR RIGHT
"A_2501_BZS16_17_I1"	I 517.7	BOOL	// BELT MONITOR LEFT
"A_2502_BZS13_I1"	I 518.2	BOOL	// DISCHARGE CHUTE PARKING POSITION
"A_2502_BZS14_I1"	I 518.3	BOOL	// DISCHARGE CHUTE LEFT SIDE
"A_2502_BZS15_I1"	I 518.4	BOOL	// DISCHARGE CHUTE RIGHT SIDE
"A_2512_BZS12_I1"	I 540.0	BOOL	// SPRINKING WATER LINE 1 OPENED
"A_2512_BZS11_I1"	I 540.1	BOOL	// SPRINKING WATER LINE 1 CLOSED
"A_2512_BZS22_I1"	I 540.2	BOOL	// SPRINKING WATER LINE 2 OPENED
"A_2512_BZS21_I1"	I 540.3	BOOL	// SPRINKING WATER LINE 2 CLOSED
"A_2511_KCL01_I1"	I 540.4	BOOL	// SCREW ON
"A_2511_KCL01_I2"	I 540.5	BOOL	// SCREW OFF
"A_2511_KCL01_I3"	I 540.6	BOOL	// DRIVE FORWARD SLOWLY
"A_2511_KCL01_I4"	I 540.7	BOOL	// DRIVE BACKWARD SLOWLY
"A_2511_KCL01_I5"	I 541.0	BOOL	// DRIVE FORWARD FASTER
"A_2511_KCL01_I6"	I 541.1	BOOL	// DRIVE BACKWARD FASTER
"A_2511_BZS44_I1"	I 541.2	BOOL	// TRAVELING DRIVE STOP LEFT SIDE
"A_2511_BZS46_I1"	I 541.3	BOOL	// TRAVELING DRIVE STOP RIGHT SIDE
"A_25_K738R1_I1"	I 542.0	BOOL	// FUSE SWITCH OFF +M251
"A_25_A408Z1_I1"	I 542.1	BOOL	// BUMPER SWITCHED-OFF
"A_2599_SHE03_I1"	I 542.2	BOOL	// EMERGENCY-STOP 1 MACHINE BMKE
"A_2599_SHE06_I1"	I 542.3	BOOL	// EMERGENCY-STOP 2 MACHINE BMKE
"A_2511_QYS43_I1"	I 542.4	BOOL	// TRAVELING DRIVE SAFETY STLEFT SIDE
"A_2511_QYS45_I1"	I 542.5	BOOL	// TRAVELING DRIVE SAFETY STRIGHT SIDE
"A_2599_SHE20_I1"	I 542.6	BOOL	// CABLE PULL SWITCH RIGHT
"A_2599_SHE21_I1"	I 542.7	BOOL	// CABLE PULL SWITCH LEFT
"A_2511_BZS22_I1"	I 543.0	BOOL	// COUPLING DRIVE UNLOCKED
"A_2511_BZS23_I1"	I 543.1	BOOL	// COUPLING DRIVE LOCKED
"A_2511_BZS26_I1"	I 543.2	BOOL	// COUPLING DRIVE UNLOCKED
"A_2511_BZS27_I1"	I 543.3	BOOL	// COUPLING DRIVE LOCKED
"A_2511_BZS32_I1"	I 543.4	BOOL	// COUPLING DRIVE UNLOCKED
"A_2511_BZS33_I1"	I 543.5	BOOL	// COUPLING DRIVE LOCKED
"A_2511_BZS36_I1"	I 543.6	BOOL	// COUPLING DRIVE UNLOCKED
"A_2511_BZS37_I1"	I 543.7	BOOL	// COUPLING DRIVE LOCKED
"A_2515_KCL01_I1"	I 560.0	BOOL	// BACKWALL LIFTING
"A_2515_KCL01_I2"	I 560.1	BOOL	// BACKWALL LOWERING
"A_2515_KCL01_I3"	I 560.2	BOOL	// UNCOUPLE
"A_2515_KCL01_I4"	I 560.3	BOOL	// COUPLE
"A_2515_KCL01_I5"	I 560.4	BOOL	// WALL LOCKING
"A_2515_KCL01_I6"	I 560.5	BOOL	// WALL UNLOCKING
"A_2515_KCL01_I7"	I 560.6	BOOL	// HORIZONTAL SCREW ON
"A_2515_KCL01_I8"	I 560.7	BOOL	// DIAGONAL SCREW ON
"A_2515_KCL01_I9"	I 561.0	BOOL	// SCREW STOP
"A_2515_BSA12_I1"	I 561.2	BOOL	// ZERO SPEED MONITOR HORIZONTAL SCREW
"A_2515_BSA17_I1"	I 561.3	BOOL	// ZERO SPEED MONITOR LIFTING SCREW
"A_25_K838R1_I1"	I 562.0	BOOL	// FUSE SWITCH OFF +M252
"A_2599_SHE04_I1"	I 562.1	BOOL	// EMERGENCY-STOP 1 MACHINE DBFL
"A_2599_SHE05_I1"	I 562.2	BOOL	// EMERGENCY-STOP 2 MACHINE DBFL
"A_2599_SHE08_I1"	I 562.3	BOOL	// EMERGENCY-STOP 3 MACHINE DBFL
"A_2515_QYS18_I1"	I 562.4	BOOL	// CLEANING FLAP 1
"A_2515_QYS19_I1"	I 562.5	BOOL	// CLEANING FLAP 2
"A_2515_BTT11_I1"	I 562.6	BOOL	// THERMISTOR HORIZONTAL SCREW
"A_2515_BTT15_I1"	I 562.7	BOOL	// THERMISTOR LIFTING SCREW
"A_2515_BZS42_I1"	I 563.0	BOOL	// COUPLING DRIVE UNLOCKED
"A_2515_BZS43_I1"	I 563.1	BOOL	// COUPLING DRIVE LOCKED
"A_2515_BZS46_I1"	I 563.2	BOOL	// COUPLING DRIVE UNLOCKED
"A_2515_BZS47_I1"	I 563.3	BOOL	// COUPLING DRIVE LOCKED
"A_2550_MXZ01_I1"	I 564.0	BOOL	// AIR-FLAP 1 OPEN
"A_2550_MXZ01_I2"	I 564.1	BOOL	// AIR-FLAP 1 CLOSE
"A_2550_BZS01_I1"	I 564.2	BOOL	// AIR-FLAP 1 CLOSED
"A_2550_BZS02_I1"	I 564.3	BOOL	// AIR-FLAP 1 OPENED
"A_2551_MXZ01_I1"	I 564.4	BOOL	// AIR-FLAP 2 OPEN
"A_2551_MXZ01_I2"	I 564.5	BOOL	// AIR-FLAP 2 CLOSE
"A_2551_BZS01_I1"	I 564.6	BOOL	// AIR-FLAP 2 CLOSED
"A_2551_BZS02_I1"	I 564.7	BOOL	// AIR-FLAP 2 OPENED
"A_2552_MXZ01_I1"	I 565.0	BOOL	// AIR-FLAP 3 OPEN
"A_2552_MXZ01_I2"	I 565.1	BOOL	// AIR-FLAP 3 CLOSE
"A_2552_BZS01_I1"	I 565.2	BOOL	// AIR-FLAP 3 CLOSED
"A_2552_BZS02_I1"	I 565.3	BOOL	// AIR-FLAP 3 OPENED
"A_2554_MXZ01_I1"	I 565.4	BOOL	// WATER PUMP 1
"A_2555_MXZ01_I1"	I 565.5	BOOL	// WATER PUMP 2
"A_2560_MXZ01_I1"	I 565.6	BOOL	// GERM FAN 1
"A_2560_MXZ02_I1"	I 565.7	BOOL	// GERM FAN 2
"A_26_A040Z1_I1"	I 600.0	BOOL	// POWER SUPPLY FAILURE +C26
"A_26_S_H097Z1_I1"	I 600.1	BOOL	// OPERATING ON +C26
"A_26_K091Z1_I1"	I 600.2	BOOL	// FUSE SWITCH OFF +C26
"A_26_A097Z1_I1"	I 600.3	BOOL	// EMERGENCY-STOP +C26
"A_26_A098Z1_I1"	I 600.4	BOOL	// EMERGENCY-STOP +M261/M262
"A_26_Q390Z1_I1"	I 600.5	BOOL	// POWER SUPPLY MACHINE BMKE
"A_26_Q445Z1_I1"	I 600.6	BOOL	// POWER SUPPLY MACHINE DBFL
"A_26_D1B065_I1"	I 600.7	BOOL	// CONTROL 24VDC LIMIT SWITCHES WAY
"A_2699_SHE01_I1"	I 601.0	BOOL	// EMERGENCY-OFF CUSTOMER
"A_2699_SHE02_I1"	I 601.1	BOOL	// EMERGENCY-OFF CUSTOMER
"A_26_A700Z1_I1"	I 601.4	BOOL	// POWER CIRCUIT CABLE CHAIN
"A_26_A106Z1_I1"	I 601.5	BOOL	// EMERGENCY-STOP FROM +C25
"A_26_A800Z1_I1"	I 601.6	BOOL	// POWER CIRCUIT CABLE CHAIN
"A_2601_MXZ01_I1"	I 602.0	BOOL	// BELT CONVEYOR
"A_2602_YMXZ01_I1"	I 602.1	BOOL	// CHUTE DRIVE LEFT SIDE
"A_2602_YMXZ01_I2"	I 602.2	BOOL	// CHUTE DRIVE RIGHT SIDE
"A_2611_MXZ41_I1"	I 603.0	BOOL	// TRAVELING DRIVE
"A_2611_MXZ61_I1"	I 603.2	BOOL	// TURNING SCREW DRIVE 1
"A_2611_MXZ62_I1"	I 603.3	BOOL	// TURNING SCREW DRIVE 2
"A_2611_MXZ63_I1"	I 603.4	BOOL	// TURNING SCREW DRIVE 3
"A_2611_MXZ64_I1"	I 603.5	BOOL	// TURNING SCREW DRIVE 4
"A_2611_MXZ65_I1"	I 603.6	BOOL	// TURNING SCREW DRIVE 5
"A_2611_MXZ66_I1"	I 603.7	BOOL	// TURNING SCREW DRIVE 6
"A_2611_MXZ67_I1"	I 604.0	BOOL	// TURNING SCREW DRIVE 7
"A_2611_MXZ68_I1"	I 604.1	BOOL	// TURNING SCREW DRIVE 8
"A_2611_MXZ69_I1"	I 604.2	BOOL	// TURNING SCREW DRIVE 9
"A_2611_MXZ70_I1"	I 604.3	BOOL	// TURNING SCREW DRIVE 10
"A_2611_MXZ71_I1"	I 604.4	BOOL	// TURNING SCREW DRIVE 11
"A_2611_MXZ72_I1"	I 604.5	BOOL	// TURNING SCREW DRIVE 12
"A_2611_MXZ73_I1"	I 604.6	BOOL	// TURNING SCREW DRIVE 13
"A_2601_SHE20_I1"	I 605.0	BOOL	// CABLE PULL SWITCH RIGHT 1
"A_2601_SHE21_I1"	I 605.1	BOOL	// CABLE PULL SWITCH RIGHT 2
"A_2601_SHE22_I1"	I 605.2	BOOL	// CABLE PULL SWITCH LEFT 1
"A_2601_SHE23_I1"	I 605.3	BOOL	// CABLE PULL SWITCH LEFT 2
"A_2602_QYS21_I1"	I 605.5	BOOL	// DISCHARGE CHUTE LEFT SIDE
"A_2602_QYS22_I1"	I 605.6	BOOL	// DISCHARGE CHUTE RIGHT SIDE
"A_2615_MXZ11_I1"	I 608.0	BOOL	// HORIZONTAL SCREW
"A_2615_MXZ15_I1"	I 608.2	BOOL	// LIFTING SCREW
"A_2615_MXZ21_I1"	I 608.3	BOOL	// LIFTING DEVICE DOWN
"A_2615_MXZ21_I2"	I 608.4	BOOL	// LIFTING DEVICE UP
"A_26_A458Z1_I1"	I 610.0	BOOL	// CLEANING FLAP 1/2
"A_2615_BZS22_I1"	I 610.6	BOOL	// LIFTING DEVICE DOWN
"A_2615_BZS23_I1"	I 610.7	BOOL	// LIFTING DEVICE END POSITION TOP
"A_2645_QXV21_I1"	I 616.0	BOOL	// RUNNING COOLING UNIT GERMINATING
"A_2645_QXV31_I1"	I 616.1	BOOL	// RUNNING COOLING UNIT GERMINATING
"A_2616_BZS12_I1"	I 616.4	BOOL	// SPRINKING WATER LINE OPENED
"A_2616_BZS11_I1"	I 616.5	BOOL	// SPRINKING WATER LINE CLOSED
"A_2631_BZS12_I1"	I 617.2	BOOL	// VALVE HUMIDIFICATION OPENED
"A_2631_BZS11_I1"	I 617.3	BOOL	// VALVE HUMIDIFICATION CLOSED
"A_2601_BSA13_I1"	I 617.4	BOOL	// SPEED CONTROL
"A_2601_BZS14_15_I1"	I 617.6	BOOL	// BELT MONITOR RIGHT
"A_2601_BZS16_17_I1"	I 617.7	BOOL	// BELT MONITOR LEFT
"A_2602_BZS13_I1"	I 618.2	BOOL	// DISCHARGE CHUTE PARKING POSITION
"A_2602_BZS14_I1"	I 618.3	BOOL	// DISCHARGE CHUTE LEFT SIDE
"A_2602_BZS15_I1"	I 618.4	BOOL	// DISCHARGE CHUTE RIGHT SIDE
"A_2612_BZS12_I1"	I 640.0	BOOL	// SPRINKING WATER LINE 1 OPENED
"A_2612_BZS11_I1"	I 640.1	BOOL	// SPRINKING WATER LINE 1 CLOSED
"A_2612_BZS22_I1"	I 640.2	BOOL	// SPRINKING WATER LINE 2 OPENED
"A_2612_BZS21_I1"	I 640.3	BOOL	// SPRINKING WATER LINE 2 CLOSED
"A_2611_KCL01_I1"	I 640.4	BOOL	// SCREW ON
"A_2611_KCL01_I2"	I 640.5	BOOL	// SCREW OFF
"A_2611_KCL01_I3"	I 640.6	BOOL	// DRIVE FORWARD SLOWLY
"A_2611_KCL01_I4"	I 640.7	BOOL	// DRIVE BACKWARD SLOWLY
"A_2611_KCL01_I5"	I 641.0	BOOL	// DRIVE FORWARD FASTER
"A_2611_KCL01_I6"	I 641.1	BOOL	// DRIVE BACKWARD FASTER
"A_2611_BZS44_I1"	I 641.2	BOOL	// TRAVELING DRIVE STOP LEFT SIDE
"A_2611_BZS46_I1"	I 641.3	BOOL	// TRAVELING DRIVE STOP RIGHT SIDE
"A_26_K738R1_I1"	I 642.0	BOOL	// FUSE SWITCH OFF +M261
"A_26_A408Z1_I1"	I 642.1	BOOL	// BUMPER SWITCHED-OFF
"A_2699_SHE03_I1"	I 642.2	BOOL	// EMERGENCY-STOP 1 MACHINE BMKE
"A_2699_SHE06_I1"	I 642.3	BOOL	// EMERGENCY-STOP 2 MACHINE BMKE
"A_2611_QYS43_I1"	I 642.4	BOOL	// TRAVELING DRIVE SAFETY STLEFT SIDE
"A_2611_QYS45_I1"	I 642.5	BOOL	// TRAVELING DRIVE SAFETY STRIGHT SIDE
"A_2699_SHE20_I1"	I 642.6	BOOL	// CABLE PULL SWITCH RIGHT
"A_2699_SHE21_I1"	I 642.7	BOOL	// CABLE PULL SWITCH LEFT
"A_2611_BZS22_I1"	I 643.0	BOOL	// COUPLING DRIVE UNLOCKED
"A_2611_BZS23_I1"	I 643.1	BOOL	// COUPLING DRIVE LOCKED
"A_2611_BZS26_I1"	I 643.2	BOOL	// COUPLING DRIVE UNLOCKED
"A_2611_BZS27_I1"	I 643.3	BOOL	// COUPLING DRIVE LOCKED
"A_2611_BZS32_I1"	I 643.4	BOOL	// COUPLING DRIVE UNLOCKED
"A_2611_BZS33_I1"	I 643.5	BOOL	// COUPLING DRIVE LOCKED
"A_2611_BZS36_I1"	I 643.6	BOOL	// COUPLING DRIVE UNLOCKED
"A_2611_BZS37_I1"	I 643.7	BOOL	// COUPLING DRIVE LOCKED
"A_2615_KCL01_I1"	I 660.0	BOOL	// BACKWALL LIFTING
"A_2615_KCL01_I2"	I 660.1	BOOL	// BACKWALL LOWERING
"A_2615_KCL01_I3"	I 660.2	BOOL	// UNCOUPLE
"A_2615_KCL01_I4"	I 660.3	BOOL	// COUPLE
"A_2615_KCL01_I5"	I 660.4	BOOL	// WALL LOCKING
"A_2615_KCL01_I6"	I 660.5	BOOL	// WALL UNLOCKING
"A_2615_KCL01_I7"	I 660.6	BOOL	// HORIZONTAL SCREW ON
"A_2615_KCL01_I8"	I 660.7	BOOL	// DIAGONAL SCREW ON
"A_2615_KCL01_I9"	I 661.0	BOOL	// SCREW STOP
"A_2615_BSA12_I1"	I 661.2	BOOL	// ZERO SPEED MONITOR HORIZONTAL SCREW
"A_2615_BSA17_I1"	I 661.3	BOOL	// ZERO SPEED MONITOR LIFTING SCREW
"A_26_K838R1_I1"	I 662.0	BOOL	// FUSE SWITCH OFF +M262
"A_2699_SHE04_I1"	I 662.1	BOOL	// EMERGENCY-STOP 1 MACHINE DBFL
"A_2699_SHE05_I1"	I 662.2	BOOL	// EMERGENCY-STOP 2 MACHINE DBFL
"A_2699_SHE08_I1"	I 662.3	BOOL	// EMERGENCY-STOP 3 MACHINE DBFL
"A_2615_QYS18_I1"	I 662.4	BOOL	// CLEANING FLAP 1
"A_2615_QYS19_I1"	I 662.5	BOOL	// CLEANING FLAP 2
"A_2615_BTT11_I1"	I 662.6	BOOL	// THERMISTOR HORIZONTAL SCREW
"A_2615_BTT15_I1"	I 662.7	BOOL	// THERMISTOR LIFTING SCREW
"A_2615_BZS42_I1"	I 663.0	BOOL	// COUPLING DRIVE UNLOCKED
"A_2615_BZS43_I1"	I 663.1	BOOL	// COUPLING DRIVE LOCKED
"A_2615_BZS46_I1"	I 663.2	BOOL	// COUPLING DRIVE UNLOCKED
"A_2615_BZS47_I1"	I 663.3	BOOL	// COUPLING DRIVE LOCKED
"A_2650_MXZ01_I1"	I 664.0	BOOL	// AIR-FLAP 1 OPEN
"A_2650_MXZ01_I2"	I 664.1	BOOL	// AIR-FLAP 1 CLOSE
"A_2650_BZS01_I1"	I 664.2	BOOL	// AIR-FLAP 1 CLOSED
"A_2650_BZS02_I1"	I 664.3	BOOL	// AIR-FLAP 1 OPENED
"A_2651_MXZ01_I1"	I 664.4	BOOL	// AIR-FLAP 2 OPEN
"A_2651_MXZ01_I2"	I 664.5	BOOL	// AIR-FLAP 2 CLOSE
"A_2651_BZS01_I1"	I 664.6	BOOL	// AIR-FLAP 2 CLOSED
"A_2651_BZS02_I1"	I 664.7	BOOL	// AIR-FLAP 2 OPENED
"A_2652_MXZ01_I1"	I 665.0	BOOL	// AIR-FLAP 3 OPEN
"A_2652_MXZ01_I2"	I 665.1	BOOL	// AIR-FLAP 3 CLOSE
"A_2652_BZS01_I1"	I 665.2	BOOL	// AIR-FLAP 3 CLOSED
"A_2652_BZS02_I1"	I 665.3	BOOL	// AIR-FLAP 3 OPENED
"A_2654_MXZ01_I1"	I 665.4	BOOL	// WATER PUMP 1
"A_2655_MXZ01_I1"	I 665.5	BOOL	// WATER PUMP 2
"A_2660_MXZ01_I1"	I 665.6	BOOL	// GERM FAN 1
"A_2660_MXZ02_I1"	I 665.7	BOOL	// GERM FAN 2
"A_27_A040Z1_I1"	I 700.0	BOOL	// POWER SUPPLY FAILURE +C27
"A_27_S_H097Z1_I1"	I 700.1	BOOL	// OPERATING ON +C27
"A_27_K091Z1_I1"	I 700.2	BOOL	// FUSE SWITCH OFF +C27
"A_27_A097Z1_I1"	I 700.3	BOOL	// EMERGENCY-STOP +C27
"A_27_A098Z1_I1"	I 700.4	BOOL	// EMERGENCY-STOP +M271/M272
"A_27_Q390Z1_I1"	I 700.5	BOOL	// POWER SUPPLY MACHINE BMKE
"A_27_Q445Z1_I1"	I 700.6	BOOL	// POWER SUPPLY MACHINE DBFL
"A_27_D1B065_I1"	I 700.7	BOOL	// CONTROL 24VDC LIMIT SWITCHES WAY
"A_2799_SHE01_I1"	I 701.0	BOOL	// EMERGENCY-OFF CUSTOMER
"A_2799_SHE02_I1"	I 701.1	BOOL	// EMERGENCY-OFF CUSTOMER
"A_27_A700Z1_I1"	I 701.4	BOOL	// POWER CIRCUIT CABLE CHAIN
"A_27_A106Z1_I1"	I 701.5	BOOL	// EMERGENCY-STOP FROM +C28
"A_27_A800Z1_I1"	I 701.6	BOOL	// POWER CIRCUIT CABLE CHAIN
"A_2701_MXZ01_I1"	I 702.0	BOOL	// BELT CONVEYOR
"A_2702_YMXZ01_I1"	I 702.1	BOOL	// CHUTE DRIVE LEFT SIDE
"A_2702_YMXZ01_I2"	I 702.2	BOOL	// CHUTE DRIVE RIGHT SIDE
"A_2711_MXZ41_I1"	I 703.0	BOOL	// TRAVELING DRIVE
"A_2711_MXZ61_I1"	I 703.2	BOOL	// TURNING SCREW DRIVE 1
"A_2711_MXZ62_I1"	I 703.3	BOOL	// TURNING SCREW DRIVE 2
"A_2711_MXZ63_I1"	I 703.4	BOOL	// TURNING SCREW DRIVE 3
"A_2711_MXZ64_I1"	I 703.5	BOOL	// TURNING SCREW DRIVE 4
"A_2711_MXZ65_I1"	I 703.6	BOOL	// TURNING SCREW DRIVE 5
"A_2711_MXZ66_I1"	I 703.7	BOOL	// TURNING SCREW DRIVE 6
"A_2711_MXZ67_I1"	I 704.0	BOOL	// TURNING SCREW DRIVE 7
"A_2711_MXZ68_I1"	I 704.1	BOOL	// TURNING SCREW DRIVE 8
"A_2711_MXZ69_I1"	I 704.2	BOOL	// TURNING SCREW DRIVE 9
"A_2711_MXZ70_I1"	I 704.3	BOOL	// TURNING SCREW DRIVE 10
"A_2711_MXZ71_I1"	I 704.4	BOOL	// TURNING SCREW DRIVE 11
"A_2711_MXZ72_I1"	I 704.5	BOOL	// TURNING SCREW DRIVE 12
"A_2711_MXZ73_I1"	I 704.6	BOOL	// TURNING SCREW DRIVE 13
"A_2701_SHE20_I1"	I 705.0	BOOL	// CABLE PULL SWITCH RIGHT 1
"A_2701_SHE21_I1"	I 705.1	BOOL	// CABLE PULL SWITCH RIGHT 2
"A_2701_SHE22_I1"	I 705.2	BOOL	// CABLE PULL SWITCH LEFT 1
"A_2701_SHE23_I1"	I 705.3	BOOL	// CABLE PULL SWITCH LEFT 2
"A_2702_QYS21_I1"	I 705.5	BOOL	// DISCHARGE CHUTE LEFT SIDE
"A_2702_QYS22_I1"	I 705.6	BOOL	// DISCHARGE CHUTE RIGHT SIDE
"A_2715_MXZ11_I1"	I 708.0	BOOL	// HORIZONTAL SCREW
"A_2715_MXZ15_I1"	I 708.2	BOOL	// LIFTING SCREW
"A_2715_MXZ21_I1"	I 708.3	BOOL	// LIFTING DEVICE DOWN
"A_2715_MXZ21_I2"	I 708.4	BOOL	// LIFTING DEVICE UP
"A_27_A458Z1_I1"	I 710.0	BOOL	// CLEANING FLAP 1/2
"A_2715_BZS22_I1"	I 710.6	BOOL	// LIFTING DEVICE DOWN
"A_2715_BZS23_I1"	I 710.7	BOOL	// LIFTING DEVICE END POSITION TOP
"A_2745_QXV21_I1"	I 716.0	BOOL	// RUNNING COOLING UNIT GERMINATING
"A_2745_QXV31_I1"	I 716.1	BOOL	// RUNNING COOLING UNIT GERMINATING
"A_2716_BZS12_I1"	I 716.4	BOOL	// SPRINKING WATER LINE OPENED
"A_2716_BZS11_I1"	I 716.5	BOOL	// SPRINKING WATER LINE CLOSED
"A_2731_BZS12_I1"	I 717.2	BOOL	// VALVE HUMIDIFICATION OPENED
"A_2731_BZS11_I1"	I 717.3	BOOL	// VALVE HUMIDIFICATION CLOSED
"A_2701_BSA13_I1"	I 717.4	BOOL	// SPEED CONTROL
"A_2701_BZS14_15_I1"	I 717.6	BOOL	// BELT MONITOR RIGHT
"A_2701_BZS16_17_I1"	I 717.7	BOOL	// BELT MONITOR LEFT
"A_2702_BZS13_I1"	I 718.2	BOOL	// DISCHARGE CHUTE PARKING POSITION
"A_2702_BZS14_I1"	I 718.3	BOOL	// DISCHARGE CHUTE LEFT SIDE
"A_2702_BZS15_I1"	I 718.4	BOOL	// DISCHARGE CHUTE RIGHT SIDE
"A_2712_BZS12_I1"	I 740.0	BOOL	// SPRINKING WATER LINE 1 OPENED
"A_2712_BZS11_I1"	I 740.1	BOOL	// SPRINKING WATER LINE 1 CLOSED
"A_2712_BZS22_I1"	I 740.2	BOOL	// SPRINKING WATER LINE 2 OPENED
"A_2712_BZS21_I1"	I 740.3	BOOL	// SPRINKING WATER LINE 2 CLOSED
"A_2711_KCL01_I1"	I 740.4	BOOL	// SCREW ON
"A_2711_KCL01_I2"	I 740.5	BOOL	// SCREW OFF
"A_2711_KCL01_I3"	I 740.6	BOOL	// DRIVE FORWARD SLOWLY
"A_2711_KCL01_I4"	I 740.7	BOOL	// DRIVE BACKWARD SLOWLY
"A_2711_KCL01_I5"	I 741.0	BOOL	// DRIVE FORWARD FASTER
"A_2711_KCL01_I6"	I 741.1	BOOL	// DRIVE BACKWARD FASTER
"A_2711_BZS44_I1"	I 741.2	BOOL	// TRAVELING DRIVE STOP LEFT SIDE
"A_2711_BZS46_I1"	I 741.3	BOOL	// TRAVELING DRIVE STOP RIGHT SIDE
"A_27_K738R1_I1"	I 742.0	BOOL	// FUSE SWITCH OFF +M271
"A_27_A408Z1_I1"	I 742.1	BOOL	// BUMPER SWITCHED-OFF
"A_2799_SHE03_I1"	I 742.2	BOOL	// EMERGENCY-STOP 1 MACHINE BMKE
"A_2799_SHE06_I1"	I 742.3	BOOL	// EMERGENCY-STOP 2 MACHINE BMKE
"A_2711_QYS43_I1"	I 742.4	BOOL	// TRAVELING DRIVE SAFETY STLEFT SIDE
"A_2711_QYS45_I1"	I 742.5	BOOL	// TRAVELING DRIVE SAFETY STRIGHT SIDE
"A_2799_SHE20_I1"	I 742.6	BOOL	// CABLE PULL SWITCH RIGHT
"A_2799_SHE21_I1"	I 742.7	BOOL	// CABLE PULL SWITCH LEFT
"A_2711_BZS22_I1"	I 743.0	BOOL	// COUPLING DRIVE UNLOCKED
"A_2711_BZS23_I1"	I 743.1	BOOL	// COUPLING DRIVE LOCKED
"A_2711_BZS26_I1"	I 743.2	BOOL	// COUPLING DRIVE UNLOCKED
"A_2711_BZS27_I1"	I 743.3	BOOL	// COUPLING DRIVE LOCKED
"A_2711_BZS32_I1"	I 743.4	BOOL	// COUPLING DRIVE UNLOCKED
"A_2711_BZS33_I1"	I 743.5	BOOL	// COUPLING DRIVE LOCKED
"A_2711_BZS36_I1"	I 743.6	BOOL	// COUPLING DRIVE UNLOCKED
"A_2711_BZS37_I1"	I 743.7	BOOL	// COUPLING DRIVE LOCKED
"A_2715_KCL01_I1"	I 760.0	BOOL	// BACKWALL LIFTING
"A_2715_KCL01_I2"	I 760.1	BOOL	// BACKWALL LOWERING
"A_2715_KCL01_I3"	I 760.2	BOOL	// UNCOUPLE
"A_2715_KCL01_I4"	I 760.3	BOOL	// COUPLE
"A_2715_KCL01_I5"	I 760.4	BOOL	// WALL LOCKING
"A_2715_KCL01_I6"	I 760.5	BOOL	// WALL UNLOCKING
"A_2715_KCL01_I7"	I 760.6	BOOL	// HORIZONTAL SCREW ON
"A_2715_KCL01_I8"	I 760.7	BOOL	// DIAGONAL SCREW ON
"A_2715_KCL01_I9"	I 761.0	BOOL	// SCREW STOP
"A_2715_BSA12_I1"	I 761.2	BOOL	// ZERO SPEED MONITOR HORIZONTAL SCREW
"A_2715_BSA17_I1"	I 761.3	BOOL	// ZERO SPEED MONITOR LIFTING SCREW
"A_27_K838R1_I1"	I 762.0	BOOL	// FUSE SWITCH OFF +M272
"A_2799_SHE04_I1"	I 762.1	BOOL	// EMERGENCY-STOP 1 MACHINE DBFL
"A_2799_SHE05_I1"	I 762.2	BOOL	// EMERGENCY-STOP 2 MACHINE DBFL
"A_2799_SHE08_I1"	I 762.3	BOOL	// EMERGENCY-STOP 3 MACHINE DBFL
"A_2715_QYS18_I1"	I 762.4	BOOL	// CLEANING FLAP 1
"A_2715_QYS19_I1"	I 762.5	BOOL	// CLEANING FLAP 2
"A_2715_BTT11_I1"	I 762.6	BOOL	// THERMISTOR HORIZONTAL SCREW
"A_2715_BTT15_I1"	I 762.7	BOOL	// THERMISTOR LIFTING SCREW
"A_2715_BZS42_I1"	I 763.0	BOOL	// COUPLING DRIVE UNLOCKED
"A_2715_BZS43_I1"	I 763.1	BOOL	// COUPLING DRIVE LOCKED
"A_2715_BZS46_I1"	I 763.2	BOOL	// COUPLING DRIVE UNLOCKED
"A_2715_BZS47_I1"	I 763.3	BOOL	// COUPLING DRIVE LOCKED
"A_2750_MXZ01_I1"	I 764.0	BOOL	// AIR-FLAP 1 OPEN
"A_2750_MXZ01_I2"	I 764.1	BOOL	// AIR-FLAP 1 CLOSE
"A_2750_BZS01_I1"	I 764.2	BOOL	// AIR-FLAP 1 CLOSED
"A_2750_BZS02_I1"	I 764.3	BOOL	// AIR-FLAP 1 OPENED
"A_2751_MXZ01_I1"	I 764.4	BOOL	// AIR-FLAP 2 OPEN
"A_2751_MXZ01_I2"	I 764.5	BOOL	// AIR-FLAP 2 CLOSE
"A_2751_BZS01_I1"	I 764.6	BOOL	// AIR-FLAP 2 CLOSED
"A_2751_BZS02_I1"	I 764.7	BOOL	// AIR-FLAP 2 OPENED
"A_2752_MXZ01_I1"	I 765.0	BOOL	// AIR-FLAP 3 OPEN
"A_2752_MXZ01_I2"	I 765.1	BOOL	// AIR-FLAP 3 CLOSE
"A_2752_BZS01_I1"	I 765.2	BOOL	// AIR-FLAP 3 CLOSED
"A_2752_BZS02_I1"	I 765.3	BOOL	// AIR-FLAP 3 OPENED
"A_2754_MXZ01_I1"	I 765.4	BOOL	// WATER PUMP 1
"A_2760_MXZ01_I1"	I 765.6	BOOL	// GERM FAN 1
"A_2760_MXZ02_I1"	I 765.7	BOOL	// GERM FAN 2
"A_2755_MXZ01_I1"	I 766.5	BOOL	// WATER PUMP 2
"A_28_A040Z1_I1"	I 800.0	BOOL	// POWER SUPPLY FAILURE +C28
"A_28_S_H097Z1_I1"	I 800.1	BOOL	// OPERATING ON +C28
"A_28_K091Z1_I1"	I 800.2	BOOL	// FUSE SWITCH OFF +C28
"A_28_A097Z1_I1"	I 800.3	BOOL	// EMERGENCY-STOP +C28
"A_28_A098Z1_I1"	I 800.4	BOOL	// EMERGENCY-STOP +M281/M282
"A_28_Q390Z1_I1"	I 800.5	BOOL	// POWER SUPPLY MACHINE BMKE
"A_28_Q445Z1_I1"	I 800.6	BOOL	// POWER SUPPLY MACHINE DBFL
"A_28_D1B065_I1"	I 800.7	BOOL	// CONTROL 24VDC LIMIT SWITCHES WAY
"A_2899_SHE01_I1"	I 801.0	BOOL	// EMERGENCY-OFF CUSTOMER
"A_2899_SHE02_I1"	I 801.1	BOOL	// EMERGENCY-OFF CUSTOMER
"A_28_A700Z1_I1"	I 801.4	BOOL	// POWER CIRCUIT CABLE CHAIN
"A_28_A106Z1_I1"	I 801.5	BOOL	// EMERGENCY-STOP FROM +C27
"A_28_A800Z1_I1"	I 801.6	BOOL	// POWER CIRCUIT CABLE CHAIN
"A_2801_MXZ01_I1"	I 802.0	BOOL	// BELT CONVEYOR
"A_2802_YMXZ01_I1"	I 802.1	BOOL	// CHUTE DRIVE LEFT SIDE
"A_2802_YMXZ01_I2"	I 802.2	BOOL	// CHUTE DRIVE RIGHT SIDE
"A_2811_MXZ41_I1"	I 803.0	BOOL	// TRAVELING DRIVE
"A_2811_MXZ61_I1"	I 803.2	BOOL	// TURNING SCREW DRIVE 1
"A_2811_MXZ62_I1"	I 803.3	BOOL	// TURNING SCREW DRIVE 2
"A_2811_MXZ63_I1"	I 803.4	BOOL	// TURNING SCREW DRIVE 3
"A_2811_MXZ64_I1"	I 803.5	BOOL	// TURNING SCREW DRIVE 4
"A_2811_MXZ65_I1"	I 803.6	BOOL	// TURNING SCREW DRIVE 5
"A_2811_MXZ66_I1"	I 803.7	BOOL	// TURNING SCREW DRIVE 6
"A_2811_MXZ67_I1"	I 804.0	BOOL	// TURNING SCREW DRIVE 7
"A_2811_MXZ68_I1"	I 804.1	BOOL	// TURNING SCREW DRIVE 8
"A_2811_MXZ69_I1"	I 804.2	BOOL	// TURNING SCREW DRIVE 9
"A_2811_MXZ70_I1"	I 804.3	BOOL	// TURNING SCREW DRIVE 10
"A_2811_MXZ71_I1"	I 804.4	BOOL	// TURNING SCREW DRIVE 11
"A_2811_MXZ72_I1"	I 804.5	BOOL	// TURNING SCREW DRIVE 12
"A_2811_MXZ73_I1"	I 804.6	BOOL	// TURNING SCREW DRIVE 13
"A_2801_SHE20_I1"	I 805.0	BOOL	// CABLE PULL SWITCH RIGHT 1
"A_2801_SHE21_I1"	I 805.1	BOOL	// CABLE PULL SWITCH RIGHT 2
"A_2801_SHE22_I1"	I 805.2	BOOL	// CABLE PULL SWITCH LEFT 1
"A_2801_SHE23_I1"	I 805.3	BOOL	// CABLE PULL SWITCH LEFT 2
"A_2802_QYS21_I1"	I 805.5	BOOL	// DISCHARGE CHUTE LEFT SIDE
"A_2802_QYS22_I1"	I 805.6	BOOL	// DISCHARGE CHUTE RIGHT SIDE
"A_2815_MXZ11_I1"	I 808.0	BOOL	// HORIZONTAL SCREW
"A_2815_MXZ15_I1"	I 808.2	BOOL	// LIFTING SCREW
"A_2815_MXZ21_I1"	I 808.3	BOOL	// LIFTING DEVICE DOWN
"A_2815_MXZ21_I2"	I 808.4	BOOL	// LIFTING DEVICE UP
"A_28_A458Z1_I1"	I 810.0	BOOL	// CLEANING FLAP 1/2
"A_2815_BZS22_I1"	I 810.6	BOOL	// LIFTING DEVICE DOWN
"A_2815_BZS23_I1"	I 810.7	BOOL	// LIFTING DEVICE END POSITION TOP
"A_2845_QXV21_I1"	I 816.0	BOOL	// RUNNING COOLING UNIT GERMINATING
"A_2845_QXV31_I1"	I 816.1	BOOL	// RUNNING COOLING UNIT GERMINATING
"A_2816_BZS12_I1"	I 816.4	BOOL	// SPRINKING WATER LINE OPENED
"A_2816_BZS11_I1"	I 816.5	BOOL	// SPRINKING WATER LINE CLOSED
"A_2831_BZS12_I1"	I 817.2	BOOL	// VALVE HUMIDIFICATION OPENED
"A_2831_BZS11_I1"	I 817.3	BOOL	// VALVE HUMIDIFICATION CLOSED
"A_2801_BSA13_I1"	I 817.4	BOOL	// SPEED CONTROL
"A_2801_BZS14_15_I1"	I 817.6	BOOL	// BELT MONITOR RIGHT
"A_2801_BZS16_17_I1"	I 817.7	BOOL	// BELT MONITOR LEFT
"A_2802_BZS13_I1"	I 818.2	BOOL	// DISCHARGE CHUTE PARKING POSITION
"A_2802_BZS14_I1"	I 818.3	BOOL	// DISCHARGE CHUTE LEFT SIDE
"A_2802_BZS15_I1"	I 818.4	BOOL	// DISCHARGE CHUTE RIGHT SIDE
"A_2812_BZS12_I1"	I 840.0	BOOL	// SPRINKING WATER LINE 1 OPENED
"A_2812_BZS11_I1"	I 840.1	BOOL	// SPRINKING WATER LINE 1 CLOSED
"A_2812_BZS22_I1"	I 840.2	BOOL	// SPRINKING WATER LINE 2 OPENED
"A_2812_BZS21_I1"	I 840.3	BOOL	// SPRINKING WATER LINE 2 CLOSED
"A_2811_KCL01_I1"	I 840.4	BOOL	// SCREW ON
"A_2811_KCL01_I2"	I 840.5	BOOL	// SCREW OFF
"A_2811_KCL01_I3"	I 840.6	BOOL	// DRIVE FORWARD SLOWLY
"A_2811_KCL01_I4"	I 840.7	BOOL	// DRIVE BACKWARD SLOWLY
"A_2811_KCL01_I5"	I 841.0	BOOL	// DRIVE FORWARD FASTER
"A_2811_KCL01_I6"	I 841.1	BOOL	// DRIVE BACKWARD FASTER
"A_2811_BZS44_I1"	I 841.2	BOOL	// TRAVELING DRIVE STOP LEFT SIDE
"A_2811_BZS46_I1"	I 841.3	BOOL	// TRAVELING DRIVE STOP RIGHT SIDE
"A_28_K738R1_I1"	I 842.0	BOOL	// FUSE SWITCH OFF +M281
"A_28_A408Z1_I1"	I 842.1	BOOL	// BUMPER SWITCHED-OFF
"A_2899_SHE03_I1"	I 842.2	BOOL	// EMERGENCY-STOP 1 MACHINE BMKE
"A_2899_SHE06_I1"	I 842.3	BOOL	// EMERGENCY-STOP 2 MACHINE BMKE
"A_2811_QYS43_I1"	I 842.4	BOOL	// TRAVELING DRIVE SAFETY STLEFT SIDE
"A_2811_QYS45_I1"	I 842.5	BOOL	// TRAVELING DRIVE SAFETY STRIGHT SIDE
"A_2899_SHE20_I1"	I 842.6	BOOL	// CABLE PULL SWITCH RIGHT
"A_2899_SHE21_I1"	I 842.7	BOOL	// CABLE PULL SWITCH LEFT
"A_2811_BZS22_I1"	I 843.0	BOOL	// COUPLING DRIVE UNLOCKED
"A_2811_BZS23_I1"	I 843.1	BOOL	// COUPLING DRIVE LOCKED
"A_2811_BZS26_I1"	I 843.2	BOOL	// COUPLING DRIVE UNLOCKED
"A_2811_BZS27_I1"	I 843.3	BOOL	// COUPLING DRIVE LOCKED
"A_2811_BZS32_I1"	I 843.4	BOOL	// COUPLING DRIVE UNLOCKED
"A_2811_BZS33_I1"	I 843.5	BOOL	// COUPLING DRIVE LOCKED
"A_2811_BZS36_I1"	I 843.6	BOOL	// COUPLING DRIVE UNLOCKED
"A_2811_BZS37_I1"	I 843.7	BOOL	// COUPLING DRIVE LOCKED
"A_2815_KCL01_I1"	I 860.0	BOOL	// BACKWALL LIFTING
"A_2815_KCL01_I2"	I 860.1	BOOL	// BACKWALL LOWERING
"A_2815_KCL01_I3"	I 860.2	BOOL	// UNCOUPLE
"A_2815_KCL01_I4"	I 860.3	BOOL	// COUPLE
"A_2815_KCL01_I5"	I 860.4	BOOL	// WALL LOCKING
"A_2815_KCL01_I6"	I 860.5	BOOL	// WALL UNLOCKING
"A_2815_KCL01_I7"	I 860.6	BOOL	// HORIZONTAL SCREW ON
"A_2815_KCL01_I8"	I 860.7	BOOL	// DIAGONAL SCREW ON
"A_2815_KCL01_I9"	I 861.0	BOOL	// SCREW STOP
"A_2815_BSA12_I1"	I 861.2	BOOL	// ZERO SPEED MONITOR HORIZONTAL SCREW
"A_2815_BSA17_I1"	I 861.3	BOOL	// ZERO SPEED MONITOR LIFTING SCREW
"A_28_K838R1_I1"	I 862.0	BOOL	// FUSE SWITCH OFF +M282
"A_2899_SHE04_I1"	I 862.1	BOOL	// EMERGENCY-STOP 1 MACHINE DBFL
"A_2899_SHE05_I1"	I 862.2	BOOL	// EMERGENCY-STOP 2 MACHINE DBFL
"A_2899_SHE08_I1"	I 862.3	BOOL	// EMERGENCY-STOP 3 MACHINE DBFL
"A_2815_QYS18_I1"	I 862.4	BOOL	// CLEANING FLAP 1
"A_2815_QYS19_I1"	I 862.5	BOOL	// CLEANING FLAP 2
"A_2815_BTT11_I1"	I 862.6	BOOL	// THERMISTOR HORIZONTAL SCREW
"A_2815_BTT15_I1"	I 862.7	BOOL	// THERMISTOR LIFTING SCREW
"A_2815_BZS42_I1"	I 863.0	BOOL	// COUPLING DRIVE UNLOCKED
"A_2815_BZS43_I1"	I 863.1	BOOL	// COUPLING DRIVE LOCKED
"A_2815_BZS46_I1"	I 863.2	BOOL	// COUPLING DRIVE UNLOCKED
"A_2815_BZS47_I1"	I 863.3	BOOL	// COUPLING DRIVE LOCKED
"A_2850_MXZ01_I1"	I 864.0	BOOL	// AIR-FLAP 1 OPEN
"A_2850_MXZ01_I2"	I 864.1	BOOL	// AIR-FLAP 1 CLOSE
"A_2850_BZS01_I1"	I 864.2	BOOL	// AIR-FLAP 1 CLOSED
"A_2850_BZS02_I1"	I 864.3	BOOL	// AIR-FLAP 1 OPENED
"A_2851_MXZ01_I1"	I 864.4	BOOL	// AIR-FLAP 2 OPEN
"A_2851_MXZ01_I2"	I 864.5	BOOL	// AIR-FLAP 2 CLOSE
"A_2851_BZS01_I1"	I 864.6	BOOL	// AIR-FLAP 2 CLOSED
"A_2851_BZS02_I1"	I 864.7	BOOL	// AIR-FLAP 2 OPENED
"A_2852_MXZ01_I1"	I 865.0	BOOL	// AIR-FLAP 3 OPEN
"A_2852_MXZ01_I2"	I 865.1	BOOL	// AIR-FLAP 3 CLOSE
"A_2852_BZS01_I1"	I 865.2	BOOL	// AIR-FLAP 3 CLOSED
"A_2852_BZS02_I1"	I 865.3	BOOL	// AIR-FLAP 3 OPENED
"A_2854_MXZ01_I1"	I 865.4	BOOL	// WATER PUMP 1
"A_2855_MXZ01_I1"	I 865.5	BOOL	// WATER PUMP 2
"A_2860_MXZ01_I1"	I 865.6	BOOL	// GERM FAN 1
"A_2860_MXZ02_I1"	I 865.7	BOOL	// GERM FAN 2
"A_3111_MXZ11_I1"	I 900.0	BOOL	// UN-/LOADING SCREW DISCHARGE
"A_3111_MXZ21_I1"	I 900.1	BOOL	// LIFTING DRIVE 1 INSIDE LOWERING
"A_3111_MXZ21_I2"	I 900.2	BOOL	// LIFTING DRIVE 1 INSIDE LIFTING
"A_3111_MXZ31_I1"	I 900.3	BOOL	// LIFTING DRIVE 2 OUTSIDE LOWERING
"A_3111_MXZ31_I2"	I 900.4	BOOL	// LIFTING DRIVE 2 OUTSIDE LIFTING
"A_3111_MXZ41_I1"	I 900.5	BOOL	// TRAVELING DRIVE
"A_31_A142F2_I1"	I 900.6	BOOL	// MAIN SWITCH BMKE
"A_3135_MXZ11_I1"	I 901.0	BOOL	// LOUVER RECYCLE AIR 1 CLOSE
"A_3135_MXZ11_I2"	I 901.1	BOOL	// LOUVER RECYCLE AIR 1 OPEN
"A_3136_MXZ11_I1"	I 901.2	BOOL	// LOUVER RECYCLE AIR 2 CLOSE
"A_3136_MXZ11_I2"	I 901.3	BOOL	// LOUVER RECYCLE AIR 2 OPEN
"A_3140_MXZ11_I1"	I 901.4	BOOL	// LOUVER RECYCLE AIR 1 CLOSE
"A_3140_MXZ11_I2"	I 901.5	BOOL	// LOUVER RECYCLE AIR 1 OPEN
"A_3141_MXZ11_I1"	I 901.6	BOOL	// LOUVER RECYCLE AIR 2 CLOSE
"A_3141_MXZ11_I2"	I 901.7	BOOL	// LOUVER RECYCLE AIR 2 OPEN
"A_3145_MXZ11_I1"	I 902.0	BOOL	// LOUVER WITHERING AIR 1 CLOSE
"A_3145_MXZ11_I2"	I 902.1	BOOL	// LOUVER WITHERING AIR 1 OPEN
"A_3146_MXZ11_I1"	I 902.2	BOOL	// LOUVER WITHERING AIR 2 CLOSE
"A_3146_MXZ11_I2"	I 902.3	BOOL	// LOUVER WITHERING AIR 2 OPEN
"A_3150_MXZ11_I1"	I 902.4	BOOL	// LOUVER FRESH AIR 1 CLOSE
"A_3150_MXZ11_I2"	I 902.5	BOOL	// LOUVER FRESH AIR 1 OPEN
"A_3151_MXZ11_I1"	I 902.6	BOOL	// LOUVER FRESH AIR 2 CLOSE
"A_3151_MXZ11_I2"	I 902.7	BOOL	// LOUVER FRESH AIR 2 OPEN
"A_3152_MXZ11_I1"	I 903.0	BOOL	// LOUVER FRESH AIR 3 CLOSE
"A_3152_MXZ11_I2"	I 903.1	BOOL	// LOUVER FRESH AIR 3 OPEN
"A_3153_MXZ11_I1"	I 903.2	BOOL	// LOUVER FRESH AIR 4 CLOSE
"A_3153_MXZ11_I2"	I 903.3	BOOL	// LOUVER FRESH AIR 4 OPEN
"A_3158_MXZ11_I1"	I 903.4	BOOL	// LOUVER AIR HEATER 1 CLOSE
"A_3158_MXZ11_I2"	I 903.5	BOOL	// LOUVER AIR HEATER 1 OPEN
"A_3159_MXZ11_I1"	I 903.6	BOOL	// LOUVER AIR HEATER 2 CLOSE
"A_3159_MXZ11_I2"	I 903.7	BOOL	// LOUVER AIR HEATER 2 OPEN
"A_3101_MXZ01_I1"	I 904.0	BOOL	// OUTLET FLAP DRIVE CLOSE
"A_3101_MXZ01_I2"	I 904.1	BOOL	// OUTLET FLAP DRIVE OPEN
"A_3125_MXZ02_I1"	I 904.2	BOOL	// GETRIEBEÖLPUMPE FAN 1
"A_3126_MXZ02_I1"	I 904.3	BOOL	// GETRIEBEÖLPUMPE FAN 2
"A_3111_QYS22_I1"	I 904.4	BOOL	// LIFTING DRIVE SAFETY STOPLIFTING DRIVE 1 INSIDE
"A_3111_QYS32_I1"	I 904.5	BOOL	// LIFTING DRIVE SAFETY STOPLIFTING DRIVE 2 OUTSIDE
"A_3135_BZS14_I1"	I 904.6	BOOL	// LOUVER RECYCLE AIR 1 CLOSED
"A_3135_BZS15_I1"	I 904.7	BOOL	// LOUVER RECYCLE AIR 1 OPENED
"A_3136_BZS14_I1"	I 905.0	BOOL	// LOUVER RECYCLE AIR 2 CLOSED
"A_3136_BZS15_I1"	I 905.1	BOOL	// LOUVER RECYCLE AIR 2 OPENED
"A_3140_BZS14_I1"	I 905.2	BOOL	// LOUVER RECYCLE AIR 1 CLOSED
"A_3140_BZS15_I1"	I 905.3	BOOL	// LOUVER RECYCLE AIR 1 OPENED
"A_3141_BZS14_I1"	I 905.4	BOOL	// LOUVER RECYCLE AIR 2 CLOSED
"A_3141_BZS15_I1"	I 905.5	BOOL	// LOUVER RECYCLE AIR 2 OPENED
"A_3145_BZS14_I1"	I 905.6	BOOL	// LOUVER WITHERING AIR 1 CLOSED
"A_3145_BZS15_I1"	I 905.7	BOOL	// LOUVER WITHERING AIR 1 OPENED
"A_3146_BZS14_I1"	I 906.0	BOOL	// LOUVER WITHERING AIR 2 CLOSED
"A_3146_BZS15_I1"	I 906.1	BOOL	// LOUVER WITHERING AIR 2 OPENED
"A_3150_BZS14_I1"	I 906.2	BOOL	// LOUVER FRESH AIR 1 CLOSED
"A_3150_BZS15_I1"	I 906.3	BOOL	// LOUVER FRESH AIR 1 OPENED
"A_3151_BZS14_I1"	I 906.4	BOOL	// LOUVER FRESH AIR 2 CLOSED
"A_3151_BZS15_I1"	I 906.5	BOOL	// LOUVER FRESH AIR 2 OPENED
"A_3152_BZS14_I1"	I 907.0	BOOL	// LOUVER FRESH AIR 3 CLOSED
"A_3152_BZS15_I1"	I 907.1	BOOL	// LOUVER FRESH AIR 3 OPENED
"A_3153_BZS14_I1"	I 907.2	BOOL	// LOUVER FRESH AIR 4 CLOSED
"A_3153_BZS15_I1"	I 907.3	BOOL	// LOUVER FRESH AIR 4 OPENED
"A_3158_BZS14_I1"	I 907.4	BOOL	// LOUVER AIR HEATER 1 CLOSED
"A_3158_BZS15_I1"	I 907.5	BOOL	// LOUVER AIR HEATER 1 OPENED
"A_3159_BZS14_I1"	I 907.6	BOOL	// LOUVER AIR HEATER 2 CLOSED
"A_3159_BZS15_I1"	I 907.7	BOOL	// LOUVER AIR HEATER 2 OPENED
"A_3101_BZS04_I1"	I 908.0	BOOL	// OUTLET FLAP CLOSED
"A_3101_BZS05_I1"	I 908.1	BOOL	// OUTLET FLAP OPENED
"A_3161_KCL11_I1"	I 916.0	BOOL	// BURNER 1 ON
"A_3161_KCL11_I2"	I 916.1	BOOL	// BURNER 1 REGULATOR ON
"A_3161_KCL11_I3"	I 916.2	BOOL	// BURNER 1 ALARM SUMMARY
"A_3161_KCL11_I4"	I 916.3	BOOL	// BURNER 1 REMOTE OPERATION
"A_3161_KCL12_I1"	I 917.0	BOOL	// BURNER 2 ON
"A_3161_KCL12_I2"	I 917.1	BOOL	// BURNER 2 REGULATOR ON
"A_3161_KCL12_I3"	I 917.2	BOOL	// BURNER 2 ALARM SUMMARY
"A_3161_KCL12_I4"	I 917.3	BOOL	// BURNER 2 REMOTE OPERATION
"A_3191_BPS21_I1"	I 918.0	BOOL	// HEAT EXCHANGE PRESSURE < 15mbar
"A_3111_BZS43_I1"	I 919.0	BOOL	// TRAVELING DRIVE POSITION
"A_3115_BZS16_I1"	I 919.4	BOOL	// CLEANING FLAP CLOSED
"A_3125_BSA07_I1"	I 920.0	BOOL	// DREHZAHLÜBERWACHUNG FAN 1
"A_3126_BSA07_I1"	I 920.1	BOOL	// DREHZAHLÜBERWACHUNG FAN 2
"A_3125_BFT09_I1"	I 920.2	BOOL	// DURCHFLUSS GETRIEBEÖL FAN 1
"A_3126_BFT09_I1"	I 920.3	BOOL	// DURCHFLUSS GETRIEBEÖL FAN 2
"A_31_A040Z1_I1"	I 924.2	BOOL	// POWER SUPPLY FAILURE +C31
"A_31_S_H097Z1_I1"	I 924.4	BOOL	// OPERATING ON +C31
"A_31_K091Z1_I1"	I 924.5	BOOL	// FUSE SWITCH OFF +C31
"A_31_A097Z1_I1"	I 924.6	BOOL	// EMERGENCY-STOP +C31
"A_3111_QYS05_I1"	I 925.0	BOOL	// DOOR CLOSED
"A_3111_BLH13_I1"	I 925.1	BOOL	// PRODUCT SENSOR
"A_3111_BZS23_I1"	I 925.2	BOOL	// LIFTING DRIVE ON THE TOP LIFTING DRIVE 1 INSIDE
"A_3111_BZS33_I1"	I 925.6	BOOL	// LIFTING DRIVE ON THE TOP LIFTING DRIVE 2 OUTSIDE
"A_3115_BZS14_I1"	I 926.4	BOOL	// DISCHARGE FLAP CLOSED
"A_3115_BZS15_I1"	I 926.5	BOOL	// DISCHARGE FLAP OPENED
"A_3125_KCU04_I1"	I 926.6	BOOL	// VIBRATION MONITOR FAN 1 ALARM CONTACT
"A_3126_KCU04_I1"	I 926.7	BOOL	// VIBRATION MONITOR FAN 2 ALARM CONTACT
"A_3199_SHE01_I1"	I 927.0	BOOL	// EMERGENCY-OFF BELOW FLOOR
"A_3199_SHE02_I1"	I 927.1	BOOL	// EMERGENCY-OFF ABOVE FLOOR
"A_3199_SHE05_I1"	I 927.4	BOOL	// EMERGENCY-OFF LADDER
"A_3211_MXZ11_I1"	I 1000.0	BOOL	// UN-/LOADING SCREW DISCHARGE
"A_3211_MXZ21_I1"	I 1000.1	BOOL	// LIFTING DRIVE 1 INSIDE LOWERING
"A_3211_MXZ21_I2"	I 1000.2	BOOL	// LIFTING DRIVE 1 INSIDE LIFTING
"A_3211_MXZ31_I1"	I 1000.3	BOOL	// LIFTING DRIVE 2 OUTSIDE LOWERING
"A_3211_MXZ31_I2"	I 1000.4	BOOL	// LIFTING DRIVE 2 OUTSIDE LIFTING
"A_3211_MXZ41_I1"	I 1000.5	BOOL	// TRAVELING DRIVE
"A_32_A142F2_I1"	I 1000.6	BOOL	// MAIN SWITCH BMKE
"A_3235_MXZ11_I1"	I 1001.0	BOOL	// LOUVER RECYCLE AIR 1 CLOSE
"A_3235_MXZ11_I2"	I 1001.1	BOOL	// LOUVER RECYCLE AIR 1 OPEN
"A_3236_MXZ11_I1"	I 1001.2	BOOL	// LOUVER RECYCLE AIR 2 CLOSE
"A_3236_MXZ11_I2"	I 1001.3	BOOL	// LOUVER RECYCLE AIR 2 OPEN
"A_3240_MXZ11_I1"	I 1001.4	BOOL	// LOUVER RECYCLE AIR 1 CLOSE
"A_3240_MXZ11_I2"	I 1001.5	BOOL	// LOUVER RECYCLE AIR 1 OPEN
"A_3241_MXZ11_I1"	I 1001.6	BOOL	// LOUVER RECYCLE AIR 2 CLOSE
"A_3241_MXZ11_I2"	I 1001.7	BOOL	// LOUVER RECYCLE AIR 2 OPEN
"A_3245_MXZ11_I1"	I 1002.0	BOOL	// LOUVER WITHERING AIR 1 CLOSE
"A_3245_MXZ11_I2"	I 1002.1	BOOL	// LOUVER WITHERING AIR 1 OPEN
"A_3246_MXZ11_I1"	I 1002.2	BOOL	// LOUVER WITHERING AIR 2 CLOSE
"A_3246_MXZ11_I2"	I 1002.3	BOOL	// LOUVER WITHERING AIR 2 OPEN
"A_3250_MXZ11_I1"	I 1002.4	BOOL	// LOUVER FRESH AIR 1 CLOSE
"A_3250_MXZ11_I2"	I 1002.5	BOOL	// LOUVER FRESH AIR 1 OPEN
"A_3251_MXZ11_I1"	I 1002.6	BOOL	// LOUVER FRESH AIR 2 CLOSE
"A_3251_MXZ11_I2"	I 1002.7	BOOL	// LOUVER FRESH AIR 2 OPEN
"A_3252_MXZ11_I1"	I 1003.0	BOOL	// LOUVER FRESH AIR 3 CLOSE
"A_3252_MXZ11_I2"	I 1003.1	BOOL	// LOUVER FRESH AIR 3 OPEN
"A_3253_MXZ11_I1"	I 1003.2	BOOL	// LOUVER FRESH AIR 4 CLOSE
"A_3253_MXZ11_I2"	I 1003.3	BOOL	// LOUVER FRESH AIR 4 OPEN
"A_3258_MXZ11_I1"	I 1003.4	BOOL	// LOUVER AIR HEATER 1 CLOSE
"A_3258_MXZ11_I2"	I 1003.5	BOOL	// LOUVER AIR HEATER 1 OPEN
"A_3259_MXZ11_I1"	I 1003.6	BOOL	// LOUVER AIR HEATER 2 CLOSE
"A_3259_MXZ11_I2"	I 1003.7	BOOL	// LOUVER AIR HEATER 2 OPEN
"A_3201_MXZ01_I1"	I 1004.0	BOOL	// OUTLET FLAP DRIVE CLOSE
"A_3201_MXZ01_I2"	I 1004.1	BOOL	// OUTLET FLAP DRIVE OPEN
"A_3225_MXZ02_I1"	I 1004.2	BOOL	// GETRIEBEÖLPUMPE FAN 1
"A_3226_MXZ02_I1"	I 1004.3	BOOL	// GETRIEBEÖLPUMPE FAN 2
"A_3211_QYS22_I1"	I 1004.4	BOOL	// LIFTING DRIVE SAFETY STOPLIFTING DRIVE 1 INSIDE
"A_3211_QYS32_I1"	I 1004.5	BOOL	// LIFTING DRIVE SAFETY STOPLIFTING DRIVE 2 OUTSIDE
"A_3235_BZS14_I1"	I 1004.6	BOOL	// LOUVER RECYCLE AIR 1 CLOSED
"A_3235_BZS15_I1"	I 1004.7	BOOL	// LOUVER RECYCLE AIR 1 OPENED
"A_3236_BZS14_I1"	I 1005.0	BOOL	// LOUVER RECYCLE AIR 2 CLOSED
"A_3236_BZS15_I1"	I 1005.1	BOOL	// LOUVER RECYCLE AIR 2 OPENED
"A_3240_BZS14_I1"	I 1005.2	BOOL	// LOUVER RECYCLE AIR 1 CLOSED
"A_3240_BZS15_I1"	I 1005.3	BOOL	// LOUVER RECYCLE AIR 1 OPENED
"A_3241_BZS14_I1"	I 1005.4	BOOL	// LOUVER RECYCLE AIR 2 CLOSED
"A_3241_BZS15_I1"	I 1005.5	BOOL	// LOUVER RECYCLE AIR 2 OPENED
"A_3245_BZS14_I1"	I 1005.6	BOOL	// LOUVER WITHERING AIR 1 CLOSED
"A_3245_BZS15_I1"	I 1005.7	BOOL	// LOUVER WITHERING AIR 1 OPENED
"A_3246_BZS14_I1"	I 1006.0	BOOL	// LOUVER WITHERING AIR 2 CLOSED
"A_3246_BZS15_I1"	I 1006.1	BOOL	// LOUVER WITHERING AIR 2 OPENED
"A_3250_BZS14_I1"	I 1006.2	BOOL	// LOUVER FRESH AIR 1 CLOSED
"A_3250_BZS15_I1"	I 1006.3	BOOL	// LOUVER FRESH AIR 1 OPENED
"A_3251_BZS14_I1"	I 1006.4	BOOL	// LOUVER FRESH AIR 2 CLOSED
"A_3251_BZS15_I1"	I 1006.5	BOOL	// LOUVER FRESH AIR 2 OPENED
"A_3252_BZS14_I1"	I 1007.0	BOOL	// LOUVER FRESH AIR 3 CLOSED
"A_3252_BZS15_I1"	I 1007.1	BOOL	// LOUVER FRESH AIR 3 OPENED
"A_3253_BZS14_I1"	I 1007.2	BOOL	// LOUVER FRESH AIR 4 CLOSED
"A_3253_BZS15_I1"	I 1007.3	BOOL	// LOUVER FRESH AIR 4 OPENED
"A_3258_BZS14_I1"	I 1007.4	BOOL	// LOUVER AIR HEATER 1 CLOSED
"A_3258_BZS15_I1"	I 1007.5	BOOL	// LOUVER AIR HEATER 1 OPENED
"A_3259_BZS14_I1"	I 1007.6	BOOL	// LOUVER AIR HEATER 2 CLOSED
"A_3259_BZS15_I1"	I 1007.7	BOOL	// LOUVER AIR HEATER 2 OPENED
"A_3201_BZS04_I1"	I 1008.0	BOOL	// OUTLET FLAP CLOSED
"A_3201_BZS05_I1"	I 1008.1	BOOL	// OUTLET FLAP OPENED
"A_3261_KCL11_I1"	I 1016.0	BOOL	// BURNER 3 ON
"A_3261_KCL11_I2"	I 1016.1	BOOL	// BURNER 3 REGULATOR ON
"A_3261_KCL11_I3"	I 1016.2	BOOL	// BURNER 3 ALARM SUMMARY
"A_3261_KCL11_I4"	I 1016.3	BOOL	// BURNER 3 REMOTE OPERATION
"A_3291_BPS21_I1"	I 1018.0	BOOL	// HEAT EXCHANGE PRESSURE < 15mbar
"A_3211_BZS43_I1"	I 1019.0	BOOL	// TRAVELING DRIVE POSITION
"A_3215_BZS16_I1"	I 1019.4	BOOL	// CLEANING FLAP CLOSED
"A_3225_BSA07_I1"	I 1020.0	BOOL	// DREHZAHLÜBERWACHUNG FAN 1
"A_3226_BSA07_I1"	I 1020.1	BOOL	// DREHZAHLÜBERWACHUNG FAN 2
"A_3225_BFT09_I1"	I 1020.2	BOOL	// DURCHFLUSS GETRIEBEÖL FAN 1
"A_3226_BFT09_I1"	I 1020.3	BOOL	// DURCHFLUSS GETRIEBEÖL FAN 2
"A_32_A040Z1_I1"	I 1024.2	BOOL	// POWER SUPPLY FAILURE +C32
"A_32_S_H097Z1_I1"	I 1024.4	BOOL	// OPERATING ON +C32
"A_32_K091Z1_I1"	I 1024.5	BOOL	// FUSE SWITCH OFF +C32
"A_32_A097Z1_I1"	I 1024.6	BOOL	// EMERGENCY-STOP +C32
"A_3211_QYS05_I1"	I 1025.0	BOOL	// DOOR CLOSED
"A_3211_BLH13_I1"	I 1025.1	BOOL	// PRODUCT SENSOR
"A_3211_BZS23_I1"	I 1025.2	BOOL	// LIFTING DRIVE ON THE TOP LIFTING DRIVE 1 INSIDE
"A_3211_BZS33_I1"	I 1025.6	BOOL	// LIFTING DRIVE ON THE TOP LIFTING DRIVE 2 OUTSIDE
"A_3215_BZS14_I1"	I 1026.4	BOOL	// DISCHARGE FLAP CLOSED
"A_3215_BZS15_I1"	I 1026.5	BOOL	// DISCHARGE FLAP OPENED
"A_3225_KCU04_I1"	I 1026.6	BOOL	// VIBRATION MONITOR FAN 1 ALARM CONTACT
"A_3226_KCU04_I1"	I 1026.7	BOOL	// VIBRATION MONITOR FAN 2 ALARM CONTACT
"A_3299_SHE01_I1"	I 1027.0	BOOL	// EMERGENCY-OFF BELOW FLOOR
"A_3299_SHE02_I1"	I 1027.1	BOOL	// EMERGENCY-OFF ABOVE FLOOR
"A_3299_SHE05_I1"	I 1027.4	BOOL	// EMERGENCY-OFF LADDER
"A_19_A040Z1_I1"	I 1100.0	BOOL	// POWER SUPPLY FAILURE +C19
"A_19_S_H097Z1_I1"	I 1100.1	BOOL	// OPERATING ON +C19
"A_19_K091Z1_I1"	I 1100.2	BOOL	// FUSE SWITCH OFF +C19
"A_19_A097Z1_I1"	I 1100.3	BOOL	// EMERGENCY-STOP +C19
"A_1999_SHE01_I1"	I 1101.0	BOOL	// EMERGENCY-OFF CONVEYOR GREEN MALT
"A_1999_SHE02_I1"	I 1101.1	BOOL	// EMERGENCY-OFF CONVEYOR GREEN MALT
"A_1911_MXZ01_I1"	I 1102.0	BOOL	// BELT CONVEYOR
"A_1915_MXZ01_I1"	I 1102.1	BOOL	// BELT CONVEYOR
"A_1921_MXZ01_I1"	I 1102.2	BOOL	// BELT CONVEYOR
"A_1931_MXZ01_I1"	I 1102.3	BOOL	// BELT CONVEYOR
"A_1941_MXZ01_I1"	I 1102.4	BOOL	// BELT CONVEYOR
"A_1942_YMXZ01_I1"	I 1102.6	BOOL	// CHUTE DRIVE LEFT SIDE
"A_1942_YMXZ01_I2"	I 1102.7	BOOL	// CHUTE DRIVE RIGHT SIDE
"A_1911_SHE20_I1"	I 1104.0	BOOL	// CABLE PULL SWITCH RIGHT 1
"A_1911_SHE21_I1"	I 1104.1	BOOL	// CABLE PULL SWITCH RIGHT 2
"A_1911_SHE22_I1"	I 1104.2	BOOL	// CABLE PULL SWITCH LEFT 1
"A_1911_SHE23_I1"	I 1104.3	BOOL	// CABLE PULL SWITCH LEFT 2
"A_1915_SHE20_I1"	I 1104.4	BOOL	// CABLE PULL SWITCH RIGHT 1
"A_1915_SHE21_I1"	I 1104.5	BOOL	// CABLE PULL SWITCH RIGHT 2
"A_1915_SHE22_I1"	I 1104.6	BOOL	// CABLE PULL SWITCH LEFT 1
"A_1915_SHE23_I1"	I 1104.7	BOOL	// CABLE PULL SWITCH LEFT 2
"A_1931_SHE20_I1"	I 1105.0	BOOL	// CABLE PULL SWITCH RIGHT 1
"A_1921_SHE21_I1"	I 1105.1	BOOL	// CABLE PULL SWITCH RIGHT 2
"A_1921_SHE22_I1"	I 1105.2	BOOL	// CABLE PULL SWITCH LEFT 1
"A_1921_SHE23_I1"	I 1105.3	BOOL	// CABLE PULL SWITCH LEFT 2
"A_1942_QYS31_I1"	I 1105.6	BOOL	// DISCHARGE CHUTE LEFT SIDE
"A_1942_QYS32_I1"	I 1105.7	BOOL	// DISCHARGE CHUTE RIGHT SIDE
"A_1911_BFT07_I1"	I 1108.0	BOOL	// STOWING DETECTOR DISCHARGE
"A_1911_BSA13_I1"	I 1108.1	BOOL	// SPEED CONTROL
"A_1911_BZS14_15_I1"	I 1108.2	BOOL	// BELT MONITOR .
"A_1915_BFT07_I1"	I 1108.4	BOOL	// STOWING DETECTOR DISCHARGE
"A_1915_BSA13_I1"	I 1108.5	BOOL	// SPEED CONTROL
"A_1915_BZS14_15_I1"	I 1108.6	BOOL	// BELT MONITOR .
"A_1921_BFT07_I1"	I 1109.0	BOOL	// STOWING DETECTOR DISCHARGE
"A_1921_BSA13_I1"	I 1109.1	BOOL	// SPEED CONTROL
"A_1921_BZS14_15_I1"	I 1109.2	BOOL	// BELT MONITOR .
"A_1931_BFT07_I1"	I 1109.4	BOOL	// STOWING DETECTOR DISCHARGE
"A_1931_BSA13_I1"	I 1109.5	BOOL	// SPEED CONTROL
"A_1931_BZS14_15_I1"	I 1109.6	BOOL	// BELT MONITOR .
"A_1941_BSA13_I1"	I 1110.0	BOOL	// SPEED CONTROL
"A_1941_BFT17_I1"	I 1110.1	BOOL	// STOWING DETECTOR DISCHARGE 1
"A_1941_BFT18_I1"	I 1110.2	BOOL	// STOWING DETECTOR DISCHARGE 2
"A_1941_BFT19_I1"	I 1110.3	BOOL	// STOWING DETECTOR DISCHARGE 3
"A_1941_BFT20_I1"	I 1110.4	BOOL	// STOWING DETECTOR DISCHARGE 4
"A_1941_BFT21_I1"	I 1110.5	BOOL	// STOWING DETECTOR DISCHARGE 5
"A_1941_BFT22_I1"	I 1110.6	BOOL	// STOWING DETECTOR DISCHARGE 6
"A_1941_BFT23_I1"	I 1110.7	BOOL	// STOWING DETECTOR DISCHARGE 7
"A_1941_BFT24_I1"	I 1111.0	BOOL	// STOWING DETECTOR DISCHARGE 8
"A_1941_BZS31_32_I1"	I 1111.1	BOOL	// BELT MONITOR .
"A_1941_BZS33_34_I1"	I 1111.2	BOOL	// BELT MONITOR .
"A_1942_BZS11_I1"	I 1111.4	BOOL	// DISCHARGE CHUTE PARKING POSITION
"A_1942_BZS12_I1"	I 1111.5	BOOL	// DISCHARGE CHUTE LEFT SIDE
"A_1942_BZS13_I1"	I 1111.6	BOOL	// DISCHARGE CHUTE RIGHT SIDE
"A_1942_BZS14_I1"	I 1112.0	BOOL	// DISCHARGE CHUTE G1A
"A_1942_BZS15_I1"	I 1112.1	BOOL	// DISCHARGE CHUTE G1B
"A_1942_BZS16_I1"	I 1112.2	BOOL	// DISCHARGE CHUTE G2A
"A_1942_BZS17_I1"	I 1112.3	BOOL	// DISCHARGE CHUTE G2B
"A_1942_BZS18_I1"	I 1112.4	BOOL	// DISCHARGE CHUTE G3A
"A_1942_BZS19_I1"	I 1112.5	BOOL	// DISCHARGE CHUTE G3B
"A_1942_BZS20_I1"	I 1112.6	BOOL	// DISCHARGE CHUTE G4A
"A_1942_BZS21_I1"	I 1112.7	BOOL	// DISCHARGE CHUTE G4B
"A_1942_BZS22_I1"	I 1113.0	BOOL	// DISCHARGE CHUTE G5A
"A_1942_BZS23_I1"	I 1113.1	BOOL	// DISCHARGE CHUTE G5B
"A_1942_BZS24_I1"	I 1113.2	BOOL	// DISCHARGE CHUTE G6A
"A_1942_BZS25_I1"	I 1113.3	BOOL	// DISCHARGE CHUTE G6B
"A_1942_BZS26_I1"	I 1113.4	BOOL	// DISCHARGE CHUTE G7A
"A_1942_BZS27_I1"	I 1113.5	BOOL	// DISCHARGE CHUTE G7B
"A_1942_BZS28_I1"	I 1113.6	BOOL	// DISCHARGE CHUTE G8A
"A_1942_BZS29_I1"	I 1113.7	BOOL	// DISCHARGE CHUTE G8B
"A_29_A040Z1_I1"	I 1116.0	BOOL	// POWER SUPPLY FAILURE +C29
"A_29_S_H097Z1_I1"	I 1116.1	BOOL	// OPERATING ON +C29
"A_29_K091Z1_I1"	I 1116.2	BOOL	// FUSE SWITCH OFF +C29
"A_29_A097Z1_I1"	I 1116.3	BOOL	// EMERGENCY-STOP +C29
"A_3101_KILN0_I1"	I 1116.4	BOOL	// SIGNAL ALTE DARRE INFEEDING
"A_2999_SHE01_I1"	I 1117.0	BOOL	// EMERGENCY-OFF CONVEYOR GREEN MALT
"A_2999_SHE02_I1"	I 1117.1	BOOL	// EMERGENCY-OFF CONVEYOR GREEN MALT
"A_2911_MXZ01_I1"	I 1118.0	BOOL	// BELT CONVEYOR
"A_2914_MXZ01_I1"	I 1118.1	BOOL	// BELT CONVEYOR
"A_2917_MXZ01_I1"	I 1118.2	BOOL	// BELT CONVEYOR
"A_2920_MXZ01_I1"	I 1118.3	BOOL	// BELT CONVEYOR
"A_2923_MXZ01_I1"	I 1118.4	BOOL	// BELT CONVEYOR
"A_2926_MXZ01_I1"	I 1118.5	BOOL	// BELT CONVEYOR
"A_2929_MXZ01_I1"	I 1118.6	BOOL	// BELT CONVEYOR
"A_2932_MXZ02_I1"	I 1119.0	BOOL	// BELT CONVEYOR DRIVE 1
"A_2932_MXZ02_I2"	I 1119.1	BOOL	// BELT CONVEYOR DRIVE 2
"A_2935_MXZ01_I1"	I 1119.2	BOOL	// BELT CONVEYOR RIGHT
"A_2935_MXZ01_I2"	I 1119.3	BOOL	// BELT CONVEYOR LEFT
"A_2923_SHE20_I1"	I 1120.0	BOOL	// CABLE PULL SWITCH RIGHT
"A_2923_SHE21_I1"	I 1120.1	BOOL	// CABLE PULL SWITCH LEFT
"A_2926_SHE20_I1"	I 1120.2	BOOL	// CABLE PULL SWITCH
"A_2929_SHE20_I1"	I 1120.4	BOOL	// CABLE PULL SWITCH
"A_2932_SHE25_I1"	I 1121.0	BOOL	// CABLE PULL SWITCH
"A_2932_SHE26_I1"	I 1121.1	BOOL	// CABLE PULL SWITCH
"A_2932_SHE27_I1"	I 1121.2	BOOL	// CABLE PULL SWITCH
"A_2935_SHE20_I1"	I 1121.4	BOOL	// CABLE PULL SWITCH
"A_2911_SHE41_I1"	I 1122.0	BOOL	// CABLE PULL SWITCH RIGHT 1
"A_2911_SHE42_I1"	I 1122.1	BOOL	// CABLE PULL SWITCH RIGHT 2
"A_2911_SHE43_I1"	I 1122.2	BOOL	// CABLE PULL SWITCH LEFT 1
"A_2911_SHE44_I1"	I 1122.3	BOOL	// CABLE PULL SWITCH LEFT 2
"A_2914_SHE41_I1"	I 1122.4	BOOL	// CABLE PULL SWITCH RIGHT 1
"A_2914_SHE42_I1"	I 1122.5	BOOL	// CABLE PULL SWITCH RIGHT 2
"A_2914_SHE43_I1"	I 1122.6	BOOL	// CABLE PULL SWITCH LEFT 1
"A_2914_SHE44_I1"	I 1122.7	BOOL	// CABLE PULL SWITCH LEFT 2
"A_2917_SHE41_I1"	I 1123.0	BOOL	// CABLE PULL SWITCH RIGHT 1
"A_2917_SHE42_I1"	I 1123.1	BOOL	// CABLE PULL SWITCH RIGHT 2
"A_2917_SHE43_I1"	I 1123.2	BOOL	// CABLE PULL SWITCH LEFT 1
"A_2917_SHE44_I1"	I 1123.3	BOOL	// CABLE PULL SWITCH LEFT 2
"A_2920_SHE41_I1"	I 1123.4	BOOL	// CABLE PULL SWITCH RIGHT 1
"A_2920_SHE42_I1"	I 1123.5	BOOL	// CABLE PULL SWITCH RIGHT 2
"A_2920_SHE43_I1"	I 1123.6	BOOL	// CABLE PULL SWITCH LEFT 1
"A_2920_SHE44_I1"	I 1123.7	BOOL	// CABLE PULL SWITCH LEFT 2
"A_2911_BFT07_I1"	I 1124.0	BOOL	// STOWING DETECTOR DISCHARGE
"A_2911_BSA13_I1"	I 1124.1	BOOL	// SPEED CONTROL
"A_2911_BZS14_15_I1"	I 1124.2	BOOL	// BELT MONITOR RIGHT
"A_2911_BZS16_17_I1"	I 1124.3	BOOL	// BELT MONITOR LEFT
"A_2914_BFT07_I1"	I 1124.4	BOOL	// STOWING DETECTOR DISCHARGE
"A_2914_BSA13_I1"	I 1124.5	BOOL	// SPEED CONTROL
"A_2914_BZS14_15_I1"	I 1124.6	BOOL	// BELT MONITOR RIGHT
"A_2914_BZS16_17_I1"	I 1124.7	BOOL	// BELT MONITOR LEFT
"A_2917_BFT07_I1"	I 1125.0	BOOL	// STOWING DETECTOR DISCHARGE
"A_2917_BSA13_I1"	I 1125.1	BOOL	// SPEED CONTROL
"A_2917_BZS14_15_I1"	I 1125.2	BOOL	// BELT MONITOR RIGHT
"A_2917_BZS16_17_I1"	I 1125.3	BOOL	// BELT MONITOR LEFT
"A_2920_BFT07_I1"	I 1125.4	BOOL	// STOWING DETECTOR DISCHARGE
"A_2920_BSA13_I1"	I 1125.5	BOOL	// SPEED CONTROL
"A_2920_BZS14_15_I1"	I 1125.6	BOOL	// BELT MONITOR RIGHT
"A_2920_BZS16_17_I1"	I 1125.7	BOOL	// BELT MONITOR LEFT
"A_2923_BFT07_I1"	I 1126.0	BOOL	// STOWING DETECTOR DISCHARGE
"A_2923_BSA13_I1"	I 1126.1	BOOL	// SPEED CONTROL
"A_2923_BZS14_15_I1"	I 1126.2	BOOL	// BELT MONITOR RIGHT
"A_2923_BZS16_17_I1"	I 1126.3	BOOL	// BELT MONITOR LEFT
"A_2926_BFT07_I1"	I 1126.4	BOOL	// STOWING DETECTOR DISCHARGE
"A_2926_BSA13_I1"	I 1126.5	BOOL	// SPEED CONTROL
"A_2926_BZS14_15_I1"	I 1126.6	BOOL	// BELT MONITOR
"A_2926_BZS16_17_I1"	I 1126.7	BOOL	// BELT MONITOR
"A_2929_BFT07_I1"	I 1127.0	BOOL	// STOWING DETECTOR DISCHARGE
"A_2929_BSA13_I1"	I 1127.1	BOOL	// SPEED CONTROL
"A_2929_BZS14_15_I1"	I 1127.2	BOOL	// BELT MONITOR RIGHT
"A_2929_BZS16_17_I1"	I 1127.3	BOOL	// BELT MONITOR LEFT
"A_2932_BFT07_I1"	I 1127.4	BOOL	// STOWING DETECTOR DISCHARGE
"A_2932_BSA13_I1"	I 1127.5	BOOL	// SPEED CONTROL
"A_2932_BZS14_15_I1"	I 1127.6	BOOL	// BELT MONITOR RIGHT
"A_2932_BZS16_17_I1"	I 1127.7	BOOL	// BELT MONITOR LEFT
"A_2932_BZS18_19_I1"	I 1128.0	BOOL	// BELT MONITOR RIGHT
"A_2932_BZS20_21_I1"	I 1128.1	BOOL	// BELT MONITOR LEFT
"A_2935_BFT07_I1"	I 1128.3	BOOL	// STOWING DETECTOR DISCHARGE 1
"A_2935_BFT08_I1"	I 1128.4	BOOL	// STOWING DETECTOR DISCHARGE 2
"A_2935_BSA13_I1"	I 1128.5	BOOL	// SPEED CONTROL
"A_2935_BZS14_15_I1"	I 1128.6	BOOL	// BELT MONITOR RIGHT
"A_2935_BZS16_17_I1"	I 1128.7	BOOL	// BELT MONITOR LEFT
"A_C29_FIREALARM_I1"	I 1129.1	BOOL	// FEUERALARM-SIGNAL VOM KUNDEN
"A_39_A040Z1_I1"	I 1132.0	BOOL	// POWER SUPPLY FAILURE +C39
"A_39_S_H097Z1_I1"	I 1132.1	BOOL	// OPERATING ON +C39
"A_39_K091Z1_I1"	I 1132.2	BOOL	// FUSE SWITCH OFF +C39
"A_39_A097Z1_I1"	I 1132.3	BOOL	// EMERGENCY-STOP +C39
"A_3946_MXZ01_I1"	I 1132.4	BOOL	// FLAP BOX 3946 - RUN TO LN
"A_3946_MXZ01_I2"	I 1132.5	BOOL	// FLAP BOX 3946 - RUN TO HN
"A_3999_SHE01_I1"	I 1133.0	BOOL	// EMERGENCY-OFF CONVEYOR GREEN MALT
"A_3999_SHE02_I1"	I 1133.1	BOOL	// EMERGENCY-OFF CONVEYOR GREEN MALT
"A_3930_SHE28_I1"	I 1133.4	BOOL	// EMERGENCY-OFF ELEVATOR
"A_3930_SHE29_I1"	I 1133.5	BOOL	// EMERGENCY-OFF ELEVATOR
"A_3945_SHE28_I1"	I 1133.6	BOOL	// EMERGENCY-OFF ELEVATOR
"A_3945_SHE29_I1"	I 1133.7	BOOL	// EMERGENCY-OFF ELEVATOR
"A_3911_MXZ01_I1"	I 1134.0	BOOL	// CHAIN CONVEYOR
"A_3912_MXZ01_I1"	I 1134.1	BOOL	// OUTLET FLAP DRIVE CLOSE
"A_3912_MXZ01_I2"	I 1134.2	BOOL	// OUTLET FLAP DRIVE OPEN
"A_3921_MXZ01_I1"	I 1134.4	BOOL	// CHAIN CONVEYOR
"A_3922_MXZ01_I1"	I 1134.5	BOOL	// OUTLET FLAP DRIVE CLOSE
"A_3922_MXZ01_I2"	I 1134.6	BOOL	// OUTLET FLAP DRIVE OPEN
"A_3930_MXZ01_I1"	I 1135.0	BOOL	// ELEVATOR
"A_3935_MXZ01_I1"	I 1135.2	BOOL	// FLAP BOX DRIVE RIGHT SIDE
"A_3935_MXZ01_I2"	I 1135.3	BOOL	// FLAP BOX DRIVE LEFT SIDE
"A_3938_MXZ01_I1"	I 1135.4	BOOL	// BELT CONVEYOR
"A_3945_MXZ01_I1"	I 1135.5	BOOL	// ELEVATOR
"A_3952_MXZ01_I1"	I 1135.6	BOOL	// DISCHARGER DMBG DRIVE
"A_3955_MXZ01_I1"	I 1135.7	BOOL	// SCREW CONVEYOR DRIVE
"A_3952_XCJ20_I1"	I 1136.0	BOOL	// VALVE DMBG CLOSED
"A_3952_XCJ20_I2"	I 1136.1	BOOL	// VALVE DMBG OPENED
"A_3952_XCJ20_I3"	I 1136.2	BOOL	// VALVE DMBG CLOSED
"A_3952_XCJ20_I4"	I 1136.3	BOOL	// VALVE DMBG OPENED
"A_3960_MXZ01_I1"	I 1136.4	BOOL	// FAN DRIVE
"A_3965_MXZ01_I1"	I 1136.5	BOOL	// AIRLOCK
"A_3970_MXZ01_I1"	I 1136.6	BOOL	// AIRLOCK
"A_3912_BZS04_I1"	I 1137.0	BOOL	// OUTLET FLAP CLOSED
"A_3912_BZS05_I1"	I 1137.1	BOOL	// OUTLET FLAP OPENED
"A_3922_BZS04_I1"	I 1137.2	BOOL	// OUTLET FLAP CLOSED
"A_3922_BZS05_I1"	I 1137.3	BOOL	// OUTLET FLAP OPENED
"A_3930_BZ08CU_I1"	I 1137.4	BOOL	// NO FAILURE ELEVATOR
"A_3930_KCL01_I1"	I 1137.5	BOOL	// RESET DISTURBANCE ELEVATOR
"A_3935_BZS04_I1"	I 1138.0	BOOL	// FLAP BOX RIGHT SIDE
"A_3935_BZS05_I1"	I 1138.1	BOOL	// FLAP BOX LEFT SIDE
"A_3946_BZS02_I1"	I 1138.2	BOOL	// FLAP BOX 3946 - LN
"A_3946_BZS03_I1"	I 1138.3	BOOL	// FLAP BOX 3946 - HN
"A_3938_SHE20_I1"	I 1138.4	BOOL	// CABLE PULL SWITCH RIGHT
"A_3938_SHE21_I1"	I 1138.5	BOOL	// CABLE PULL SWITCH LEFT
"A_3945_BZ08CU_I1"	I 1138.6	BOOL	// NO FAILURE ELEVATOR
"A_3945_KCL01_I1"	I 1138.7	BOOL	// RESET DISTURBANCE ELEVATOR
"A_3930_BSA07_I1"	I 1139.0	BOOL	// SPEED CONTROL
"A_3945_BSA07_I1"	I 1139.1	BOOL	// SPEED CONTROL
"A_39_A187Z1_I1"	I 1139.4	BOOL	// EMERGENCY-STOP (3930-MXZ0ELEVATOR
"A_3930_QYS30_I1"	I 1139.5	BOOL	// EXPLOSION VENT ELEVATOR
"A_39_A227Z1_I1"	I 1139.6	BOOL	// EMERGENCY-STOP (3945-MXZ0ELEVATOR
"A_3945_QYS30_I1"	I 1139.7	BOOL	// EXPLOSION VENT ELEVATOR
"A_3956_KCL01_I1"	I 1140.6	BOOL	// EXCISTING DEGERMINATING SYSTEM IS RUNNING
"A_3911_BQS06_I1"	I 1141.0	BOOL	// STOWING DETECTOR DISCHARGE
"A_3911_BSA08_I1"	I 1141.1	BOOL	// SPEED CONTROL
"A_3921_BQS06_I1"	I 1141.2	BOOL	// STOWING DETECTOR DISCHARGE
"A_3921_BSA08_I1"	I 1141.3	BOOL	// SPEED CONTROL
"A_3930_BLH31_I1"	I 1141.5	BOOL	// STOWING DETECTOR DISCHARGE
"A_3936_BFT01_I1"	I 1141.6	BOOL	// STOWING DETECTOR DISCHARGE
"A_3938_BLH07_I1"	I 1142.0	BOOL	// STOWING DETECTOR DISCHARGE
"A_3938_BSA13_I1"	I 1142.1	BOOL	// SPEED CONTROL
"A_3938_BZS14_15_I1"	I 1142.2	BOOL	// BELT MONITOR LEFT
"A_3938_BZS16_17_I1"	I 1142.3	BOOL	// BELT MONITOR MIDDLE
"A_3938_BZS18_19_I1"	I 1142.4	BOOL	// BELT MONITOR RIGHT
"A_3975_BLH01_I1"	I 1142.6	BOOL	// VOLLMELDER SILO ASPIRATION
"A_3945_BLH31_I1"	I 1143.0	BOOL	// STOWING DETECTOR DISCHARGE
"A_3951_BLL01_I1"	I 1143.1	BOOL	// STOWING DETECTOR DISCHARGE
"A_3955_BFT09_I1"	I 1143.2	BOOL	// STOWING DETECTOR DISCHARGE
"A_3955_BSA11_I1"	I 1143.3	BOOL	// SPEED CONTROL
"A_6105_MXZ01_I1"	I 1152.0	BOOL	// ELEVATOR 6105 - STARTED
"A_6106_MXZ01_I1"	I 1152.1	BOOL	// SCREW CONV. 6106 - STARTED
"A_6107_MXZ01_I1"	I 1152.2	BOOL	// OUTLET SLIDE 6107 - CLOSING
"A_6107_MXZ01_I2"	I 1152.3	BOOL	// OUTLET SLIDE 6107 - OPENING
"A_6108_MXZ01_I1"	I 1152.4	BOOL	// OUTLET SLIDE 6108 - CLOSING
"A_6108_MXZ01_I2"	I 1152.5	BOOL	// OUTLET SLIDE 6108 - OPENING
"A_6109_MXZ01_I1"	I 1152.6	BOOL	// ROUTLET SCREW 6109 - STARTED
"A_6110_MXZ01_I1"	I 1152.7	BOOL	// ROUTLET SCREW 6110 - STARTED
"A_6111_MXZ01_I1"	I 1153.0	BOOL	// SIEVE DRIVE 6111 - STARTED
"A_6112_MXZ01_I1"	I 1153.1	BOOL	// SIEVE DRIVE 6112 - STARTED
"A_6113_MXZ01_I1"	I 1153.2	BOOL	// CHAIN CONV. 6113 - STARTED
"A_6114_MXZ01_I1"	I 1153.4	BOOL	// OUTLET SLIDE 6114 - CLOSING
"A_6114_MXZ01_I2"	I 1153.5	BOOL	// OUTLET SLIDE 6114 - OPENING
"A_6115_MXZ01_I1"	I 1153.6	BOOL	// OUTLET SLIDE 6115 - CLOSING
"A_6115_MXZ01_I2"	I 1153.7	BOOL	// OUTLET SLIDE 6115 - OPENING
"A_6116_MXZ01_I1"	I 1154.0	BOOL	// OUTLET SLIDE 6116 - CLOSING
"A_6116_MXZ01_I2"	I 1154.1	BOOL	// OUTLET SLIDE 6116 - OPENING
"A_6117_MXZ01_I1"	I 1154.2	BOOL	// OUTLET SLIDE 6117 - CLOSING
"A_6117_MXZ01_I2"	I 1154.3	BOOL	// OUTLET SLIDE 6117 - OPENING
"A_6118_MXZ01_I1"	I 1154.4	BOOL	// CHAIN CONV. 6118 - STARTED
"A_6119_MXZ01_I1"	I 1154.6	BOOL	// OUTLET SLIDE 6119 - CLOSING
"A_6119_MXZ01_I2"	I 1154.7	BOOL	// OUTLET SLIDE 6119 - OPENING
"A_6120_MXZ01_I1"	I 1155.0	BOOL	// OUTLET SLIDE 6120 - CLOSING
"A_6120_MXZ01_I2"	I 1155.1	BOOL	// OUTLET SLIDE 6120 - OPENING
"A_6121_MXZ01_I1"	I 1155.2	BOOL	// CHAIN CONV. 6121 - STARTED
"A_6151_MXZ01_I1"	I 1155.4	BOOL	// OUTLET SLIDE 6151 - CLOSING
"A_6151_MXZ01_I2"	I 1155.5	BOOL	// OUTLET SLIDE 6151 - OPENING
"A_6152_MXZ01_I1"	I 1155.6	BOOL	// OUTLET SLIDE 6152 - CLOSING
"A_6152_MXZ01_I2"	I 1155.7	BOOL	// OUTLET SLIDE 6152 - OPENING
"A_6153_MXZ01_I1"	I 1156.0	BOOL	// OUTLET SLIDE 6153 - CLOSING
"A_6153_MXZ01_I2"	I 1156.1	BOOL	// OUTLET SLIDE 6153 - OPENING
"A_6154_MXZ01_I1"	I 1156.2	BOOL	// OUTLET SLIDE 6154 - CLOSING
"A_6154_MXZ01_I2"	I 1156.3	BOOL	// OUTLET SLIDE 6154 - OPENING
"A_6155_MXZ01_I1"	I 1156.4	BOOL	// OUTLET SLIDE 6155 - CLOSING
"A_6155_MXZ01_I2"	I 1156.5	BOOL	// OUTLET SLIDE 6155 - OPENING
"A_6156_MXZ01_I1"	I 1156.6	BOOL	// OUTLET SLIDE 6156 - CLOSING
"A_6156_MXZ01_I2"	I 1156.7	BOOL	// OUTLET SLIDE 6156 - OPENING
"A_6157_MXZ01_I1"	I 1157.0	BOOL	// OUTLET SLIDE 6157 - CLOSING
"A_6157_MXZ01_I2"	I 1157.1	BOOL	// OUTLET SLIDE 6157 - OPENING
"A_6161_MXZ01_I1"	I 1157.2	BOOL	// CHAIN CONV. 6161 - STARTED
"A_6162_MXZ01_I1"	I 1157.3	BOOL	// CHAIN CONV. 6162 - STARTED
"A_6163_MXZ01_I1"	I 1157.4	BOOL	// ELEVATOR 6163 - STARTED
"A_6164_MXZ01_I1"	I 1157.5	BOOL	// SCREW CONV. 6164 - STARTED
"A_6167_MXZ01_I1"	I 1157.6	BOOL	// SAMPLER 6167 - STARTED
"A_6183_MXZ01_I1"	I 1157.7	BOOL	// AIRLOCK 6183 - STARTED
"A_6184_MXZ01_I1"	I 1158.0	BOOL	// APSIRATION FAN 6184 - STARTED
"A_6105_BQS07_I1"	I 1172.0	BOOL	// ELEVATOR 6105 - STOWING DETECTOR/ INLET
"A_6106_BSA11_I1"	I 1172.1	BOOL	// SCREW CONV. 6106 - SPEED CONTROL
"A_6111_BZS04_I1"	I 1172.2	BOOL	// SIEVE BOX 6111 - UNBALANCE
"A_6112_BZS04_I1"	I 1172.3	BOOL	// SIEVE BOX 6112 - UNBALANCE
"A_6113_BLL05_I1"	I 1172.4	BOOL	// CHAIN CONV. 6113 - PRODUCT SENSING DEV.
"A_6113_BQS06_I1"	I 1172.5	BOOL	// CHAIN CONV. 6113 - OVERFILL PROTECTION
"A_6113_BSA11_I1"	I 1172.6	BOOL	// CHAIN CONV. 6113 - SPEED CONTROL
"A_6118_BQS06_I1"	I 1172.7	BOOL	// CHAIN CONV. 6118 - OVERFILL PROTECTION
"A_6118_BSA11_I1"	I 1173.0	BOOL	// CHAIN CONV. 6118 - SPEED CONTROL
"A_6121_BQS06_I1"	I 1173.1	BOOL	// CHAIN CONV. 6121 - OVERFILL PROTECTION
"A_6121_BSA11_I1"	I 1173.2	BOOL	// CHAIN CONV. 6121 - SPEED CONTROL
"A_6131_BLH01_I1"	I 1173.4	BOOL	// HIGH LEVEL BIN 198
"A_6132_BLH01_I1"	I 1173.5	BOOL	// HIGH LEVEL BIN 197
"A_6133_BLH01_I1"	I 1173.6	BOOL	// HIGH LEVEL BIN 195
"A_6134_BLH01_I1"	I 1173.7	BOOL	// HIGH LEVEL BIN 194
"A_6135_BLH01_I1"	I 1174.0	BOOL	// HIGH LEVEL BIN 193
"A_6136_BLH01_I1"	I 1174.1	BOOL	// HIGH LEVEL BIN 192
"A_6137_BLH01_I1"	I 1174.2	BOOL	// HIGH LEVEL BIN 196
"A_6141_BLL01_I1"	I 1174.3	BOOL	// LOW LEVEL BIN 198
"A_6142_BLL01_I1"	I 1174.4	BOOL	// LOW LEVEL BIN 197
"A_6143_BLL01_I1"	I 1174.5	BOOL	// LOW LEVEL BIN 195
"A_6144_BLL01_I1"	I 1174.6	BOOL	// LOW LEVEL BIN 194
"A_6145_BLL01_I1"	I 1174.7	BOOL	// LOW LEVEL BIN 193
"A_6146_BLL01_I1"	I 1175.0	BOOL	// LOW LEVEL BIN 192
"A_6147_BLL01_I1"	I 1175.1	BOOL	// LOW LEVEL BIN 196
"A_6161_BQS06_I1"	I 1175.2	BOOL	// CHAIN CONV. 6161 - OVERFILL PROTECTION
"A_6161_BSA11_I1"	I 1175.3	BOOL	// CHAIN CONV. 6161 - SPEED CONTROL
"A_6162_BLL05_I1"	I 1175.4	BOOL	// CHAIN CONV. 6162 - PROD. SENSING DEVICE
"A_6162_BQS06_I1"	I 1175.5	BOOL	// CHAIN CONV. 6162 - OVERFILL PROTECTION
"A_6162_BSA11_I1"	I 1175.6	BOOL	// CHAIN CONV. 6162 - SPEED CONTROL
"A_6163_BQS07_I1"	I 1175.7	BOOL	// ELEVATOR 6163 - STOWING DETECTOR/ INLET
"A_6164_BSA11_I1"	I 1176.0	BOOL	// SCREW CONV. 6164 - SPEED CONTROL
"A_6165_BLH01_I1"	I 1176.1	BOOL	// HIGH LEVEL - SCALE 6165
"A_6168_BLH01_I1"	I 1176.2	BOOL	// HIGH LEVEL - BEFORE EXIST. PLANT
"A_6183_BSA11_I1"	I 1176.3	BOOL	// AIRLOCK 6183 - SPEED CONTROL
"A_6167_BLH04_I1"	I 1176.5	BOOL	// SAMPLER 6167 EXP1 - HIGH LEVEL
"A_6118_KFC10_I1"	I 1177.6	BOOL	// MVRU FILTER CONTROL - ALARM
"A_6151_KCL01_I1"	I 1178.0	BOOL	// LOCAL CONTROL - CMD OPEN
"A_6151_KCL01_I2"	I 1178.1	BOOL	// LOCAL CONTROL - CMD CLOSE
"A_6151_KCL01_I3"	I 1178.2	BOOL	// LOCAL CONTROL - CMD FAILURE RESET
"A_6152_KCL01_I1"	I 1178.4	BOOL	// LOCAL CONTROL - CMD OPEN
"A_6152_KCL01_I2"	I 1178.5	BOOL	// LOCAL CONTROL - CMD CLOSE
"A_6152_KCL01_I3"	I 1178.6	BOOL	// LOCAL CONTROL - CMD FAILURE RESET
"A_6153_KCL01_I1"	I 1179.0	BOOL	// LOCAL CONTROL - CMD OPEN
"A_6153_KCL01_I2"	I 1179.1	BOOL	// LOCAL CONTROL - CMD CLOSE
"A_6153_KCL01_I3"	I 1179.2	BOOL	// LOCAL CONTROL - CMD FAILURE RESET
"A_C41_I1"	I 1179.4	BOOL	// INTERFACE 1 - SIGNAL 1
"A_C41_I2"	I 1179.5	BOOL	// INTERFACE 1 - SIGNAL 2
"A_C41_I3"	I 1179.6	BOOL	// INTERFACE 1 - SIGNAL 3
"A_C41_I4"	I 1179.7	BOOL	// INTERFACE 1 - SIGNAL 4
"A_6105_BZ08CU_I1"	I 1180.0	BOOL	// ELEVATOR 6105 - BELT MONITOR
"A_6105_BST09_I1"	I 1180.2	BOOL	// ELEVATOR 6105 - SPEED CONTROL
"A_6105_FYX20_I1"	I 1180.3	BOOL	// ELEVATOR 6105 - EXPLOSION VENT FLAP
"A_6105_SHE38_I1"	I 1180.4	BOOL	// ELEVATOR 6105 - EMERGENCY OFF/ BOTTOM
"A_6105_SHE39_I1"	I 1180.5	BOOL	// ELEVATOR 6105 - EMERGENCY OFF/ TOP
"A_6105_SHE3XA1_I1"	I 1180.6	BOOL	// ELEVATOR 6105 - EMERGENCY OFF/ DEVICE
"A_6106_BQS09_I1"	I 1180.7	BOOL	// SCREW CONV. 6105 - STOWING DETECTOR
"A_6107_BZS04_I1"	I 1181.0	BOOL	// OUTLET SLIDE 6107 - CLOSED
"A_6107_BZS05_I1"	I 1181.1	BOOL	// OUTLET SLIDE 6107 - OPENED
"A_6108_BZS04_I1"	I 1181.2	BOOL	// OUTLET SLIDE 6108 - CLOSED
"A_6108_BZS05_I1"	I 1181.3	BOOL	// OUTLET SLIDE 6108 - OPENED
"A_6114_BZS04_I1"	I 1181.4	BOOL	// OUTLET SLIDE 6114 - CLOSED
"A_6114_BZS05_I1"	I 1181.5	BOOL	// OUTLET SLIDE 6114 - OPENED
"A_6115_BZS04_I1"	I 1181.6	BOOL	// OUTLET SLIDE 6115 - CLOSED
"A_6115_BZS05_I1"	I 1181.7	BOOL	// OUTLET SLIDE 6115 - OPENED
"A_6116_BZS04_I1"	I 1182.0	BOOL	// OUTLET SLIDE 6116 - CLOSED
"A_6116_BZS05_I1"	I 1182.1	BOOL	// OUTLET SLIDE 6116 - OPENED
"A_6117_BZS04_I1"	I 1182.2	BOOL	// OUTLET SLIDE 6117 - CLOSED
"A_6117_BZS05_I1"	I 1182.3	BOOL	// OUTLET SLIDE 6117 - OPENED
"A_6119_BZS04_I1"	I 1182.4	BOOL	// OUTLET SLIDE 6119 - CLOSED
"A_6119_BZS05_I1"	I 1182.5	BOOL	// OUTLET SLIDE 6119 - OPENED
"A_6120_BZS04_I1"	I 1182.6	BOOL	// OUTLET SLIDE 6120 - CLOSED
"A_6120_BZS05_I1"	I 1182.7	BOOL	// OUTLET SLIDE 6120 - OPENED
"A_6151_BZS04_I1"	I 1183.0	BOOL	// OUTLET SLIDE 6151 - CLOSED
"A_6151_BZS05_I1"	I 1183.1	BOOL	// OUTLET SLIDE 6151 - OPENED
"A_6152_BZS04_I1"	I 1183.2	BOOL	// OUTLET SLIDE 6152 - CLOSED
"A_6152_BZS05_I1"	I 1183.3	BOOL	// OUTLET SLIDE 6152 - OPENED
"A_6999_SHE05_I1"	I 1183.4	BOOL	// EMERGENCY STOP BUTTON 5
"A_6999_SHE06_I1"	I 1183.5	BOOL	// EMERGENCY STOP BUTTON 6
"A_6999_SHE07_I1"	I 1183.6	BOOL	// EMERGENCY STOP BUTTON 7
"A_6999_SHE08_I1"	I 1183.7	BOOL	// EMERGENCY STOP BUTTON 8
"A_6153_BZS04_I1"	I 1184.0	BOOL	// OUTLET SLIDE 6153 - CLOSED
"A_6153_BZS05_I1"	I 1184.1	BOOL	// OUTLET SLIDE 6153 - OPENED
"A_6154_BZS04_I1"	I 1184.2	BOOL	// OUTLET SLIDE 6154 - CLOSED
"A_6154_BZS05_I1"	I 1184.3	BOOL	// OUTLET SLIDE 6154 - OPENED
"A_6155_BZS04_I1"	I 1184.4	BOOL	// OUTLET SLIDE 6155 - CLOSED
"A_6155_BZS05_I1"	I 1184.5	BOOL	// OUTLET SLIDE 6155 - OPENED
"A_6156_BZS04_I1"	I 1184.6	BOOL	// OUTLET SLIDE 6156 - CLOSED
"A_6156_BZS05_I1"	I 1184.7	BOOL	// OUTLET SLIDE 6156 - OPENED
"A_6157_BZS04_I1"	I 1185.0	BOOL	// OUTLET SLIDE 6157 - CLOSED
"A_6157_BZS05_I1"	I 1185.1	BOOL	// OUTLET SLIDE 6157 - OPENED
"A_6163_BZ08CU_I1"	I 1185.2	BOOL	// ELEVATOR 6163 - BELT MONITOR
"A_6163_BST09_I1"	I 1185.4	BOOL	// ELEVATOR 6163 - SPEED CONTROL
"A_6163_FYX20_I1"	I 1185.5	BOOL	// ELEVATOR 6163 - EXPLOSION VENT FLAP
"A_6163_SHE38_I1"	I 1185.6	BOOL	// ELEVATOR 6163 - EMERGENCY OFF/ BOTTOM
"A_6163_SHE39_I1"	I 1185.7	BOOL	// ELEVATOR 6163 - EMERGENCY OFF/ TOP
"A_6163_SHE3XA1_I1"	I 1186.0	BOOL	// ELEVATOR 6163 - EMERGENCY OFF/ DEVICE
"A_6164_BQS09_I1"	I 1186.1	BOOL	// SCREW CONV. 6164 - STOWING DETECTOR
"A_6167_BZS03_I1"	I 1186.2	BOOL	// SAMPLER 6167 EXP1 - LIMIT SWITCH
"A_6118_FYX06_I1"	I 1186.3	BOOL	// MAIN FILTER - EXPLOSION VENT FLAP
"A_6999_SHE09_I1"	I 1186.4	BOOL	// EMERGENCY STOP BUTTON 9
"A_6999_SHE10_I1"	I 1186.5	BOOL	// EMERGENCY STOP BUTTON 10
"A_41_S_H097Z1_I1"	I 1187.1	BOOL	// OPERATING ON +C41
"A_41_K091Z1_I1"	I 1187.2	BOOL	// FUSE SWITCH +C41
"A_41_A097Z1_I1"	I 1187.3	BOOL	// EMERGENCY STOP - DEVICE +C41
"A_6999_SHE01_I1"	I 1187.4	BOOL	// EMERGENCY STOP BUTTON 1
"A_6999_SHE02_I1"	I 1187.5	BOOL	// EMERGENCY STOP BUTTON 2
"A_6999_SHE03_I1"	I 1187.6	BOOL	// EMERGENCY STOP BUTTON 3
"A_6999_SHE04_I1"	I 1187.7	BOOL	// EMERGENCY STOP BUTTON 4
"A_2191_BTE01_AI1"	IW 168	WORD	// AIR TEMPERATURE BELOW FLOOR
"A_2191_BTE02_AI1"	IW 170	WORD	// AIR TEMPERATURE ABOVE FLOOR
"A_2145_QXV21_AI1"	IW 172	WORD	// REGULATING VALVE ACTUEL VALUE
"A_2145_QXV31_AI1"	IW 174	WORD	// REGULATING VALVE ACTUEL VALUE
"A_2150_BEE01_AI1"	IW 176	WORD	// EXHAUST FLAP ACTUEL VALUE
"A_2111_BZS49_AI1"	IW 180	WORD	// TRAVELING DRIVE POSITION CHANNEL 1/2
"A_2151_BEE01_AI1"	IW 192	WORD	//  FRESH FLAP ACTUEL VALUE
"A_2152_BEE01_AI1"	IW 194	WORD	//  FRESH FLAP ACTUEL VALUE
"A_2191_BTE03_AI1"	IW 196	WORD	// AIR TEMPERATURE BELOW FLOOR
"A_2191_BTE04_AI1"	IW 198	WORD	// AIR TEMPERATURE ABOVE FLOOR
"A_2291_BTE01_AI1"	IW 268	WORD	// AIR TEMPERATURE BELOW FLOOR
"A_2291_BTE02_AI1"	IW 270	WORD	// AIR TEMPERATURE ABOVE FLOOR
"A_2245_QXV21_AI1"	IW 272	WORD	// REGULATING VALVE ACTUEL VALUE
"A_2245_QXV31_AI1"	IW 274	WORD	// REGULATING VALVE ACTUEL VALUE
"A_2250_BEE01_AI1"	IW 276	WORD	// EXHAUST FLAP ACTUEL VALUE
"A_2211_BZS49_AI1"	IW 280	WORD	// TRAVELING DRIVE POSITION CHANNEL 1/2
"A_2251_BEE01_AI1"	IW 292	WORD	//  FRESH FLAP ACTUEL VALUE
"A_2252_BEE01_AI1"	IW 294	WORD	//  FRESH FLAP ACTUEL VALUE
"A_2291_BTE03_AI1"	IW 296	WORD	// AIR TEMPERATURE BELOW FLOOR
"A_2291_BTE04_AI1"	IW 298	WORD	// AIR TEMPERATURE ABOVE FLOOR
"A_2391_BTE01_AI1"	IW 368	WORD	// AIR TEMPERATURE BELOW FLOOR
"A_2391_BTE02_AI1"	IW 370	WORD	// AIR TEMPERATURE ABOVE FLOOR
"A_2345_QXV21_AI1"	IW 372	WORD	// REGULATING VALVE ACTUEL VALUE
"A_2345_QXV31_AI1"	IW 374	WORD	// REGULATING VALVE ACTUEL VALUE
"A_2350_BEE01_AI1"	IW 376	WORD	// EXHAUST FLAP ACTUEL VALUE
"A_2311_BZS49_AI1"	IW 380	WORD	// TRAVELING DRIVE POSITION CHANNEL 1/2
"A_2351_BEE01_AI1"	IW 392	WORD	//  FRESH FLAP ACTUEL VALUE
"A_2352_BEE01_AI1"	IW 394	WORD	//  FRESH FLAP ACTUEL VALUE
"A_2391_BTE03_AI1"	IW 396	WORD	// AIR TEMPERATURE BELOW FLOOR
"A_2391_BTE04_AI1"	IW 398	WORD	// AIR TEMPERATURE ABOVE FLOOR
"A_2491_BTE01_AI1"	IW 468	WORD	// AIR TEMPERATURE BELOW FLOOR
"A_2491_BTE02_AI1"	IW 470	WORD	// AIR TEMPERATURE ABOVE FLOOR
"A_2445_QXV21_AI1"	IW 472	WORD	// REGULATING VALVE ACTUEL VALUE
"A_2445_QXV31_AI1"	IW 474	WORD	// REGULATING VALVE ACTUEL VALUE
"A_2450_BEE01_AI1"	IW 476	WORD	// EXHAUST FLAP ACTUEL VALUE
"A_2411_BZS49_AI1"	IW 480	WORD	// TRAVELING DRIVE POSITION CHANNEL 1/2
"A_2451_BEE01_AI1"	IW 492	WORD	//  FRESH FLAP ACTUEL VALUE
"A_2452_BEE01_AI1"	IW 494	WORD	//  FRESH FLAP ACTUEL VALUE
"A_2491_BTE03_AI1"	IW 496	WORD	// AIR TEMPERATURE BELOW FLOOR
"A_2491_BTE04_AI1"	IW 498	WORD	// AIR TEMPERATURE ABOVE FLOOR
"CPU_CopyPulse100ms"	M 1.0	BOOL	// CPU: System timing
"CPU_CopyPulse200ms"	M 1.1	BOOL	// CPU: System timing
"CPU_CopyPulse400ms"	M 1.2	BOOL	// CPU: System timing
"CPU_CopyPulse500ms"	M 1.3	BOOL	// CPU: System timing
"CPU_CopyPulse800ms"	M 1.4	BOOL	// CPU: System timing
"CPU_CopyPulse1000ms"	M 1.5	BOOL	// CPU: System timing
"CPU_CopyPulse1600ms"	M 1.6	BOOL	// CPU: System timing
"CPU_CopyPulse1800ms"	M 1.7	BOOL	// CPU: System timing
"CPU_Pulse100ms"	M 2.0	BOOL	// CPU: System timing
"CPU_Pulse200ms"	M 2.1	BOOL	// CPU: System timing
"CPU_Pulse400ms"	M 2.2	BOOL	// CPU: System timing
"CPU_Pulse500ms"	M 2.3	BOOL	// CPU: System timing
"CPU_Pulse800ms"	M 2.4	BOOL	// CPU: System timing
"CPU_Pulse1000ms"	M 2.5	BOOL	// CPU: System timing
"CPU_Pulse1600ms"	M 2.6	BOOL	// CPU: System timing
"CPU_Pulse2000ms"	M 2.7	BOOL	// CPU: System timing
"SYS_ScanA_IsOn"	M 3.1	BOOL	// SYS: Scan A is active
"SYS_ScanB_IsOn"	M 3.2	BOOL	// SYS: Scan B is active
"SYS_ScanC_IsOn"	M 3.3	BOOL	// SYS: Scan C is active
"Sys_Tick100msFromFastOB"	M 3.6	BOOL
"Sys_Tick200msFromFastOB"	M 3.7	BOOL
"SYS_Scan0_Tick100ms"	M 4.2	BOOL	// SYS_Scan0: Is every 100ms for one scan high
"SYS_Scan0_Tick200ms"	M 4.3	BOOL	// SYS_Scan0: Is every 200ms for one scan high
"SYS_Scan0_Tick500ms"	M 4.4	BOOL	// SYS_Scan0: Is every 500ms for one scan high
"SYS_Scan0_Tick1s"	M 4.5	BOOL	// SYS_Scan0: Is every 1s for one scan high
"SYS_Scan0_Tick1min"	M 4.6	BOOL	// SYS_Scan0: Is every min for one scan high
"SYS_Scan0_Tick30s"	M 4.7	BOOL	// SYS_Scan0: Is every 30s for one scan high
"SYS_ScanA_Tick200ms"	M 5.3	BOOL	// SYS_ScanA: Is every 200ms for one scan high
"SYS_ScanA_Tick500ms"	M 5.4	BOOL	// SYS_ScanA:  Is every 500ms for one scan high
"SYS_ScanA_Tick1s"	M 5.5	BOOL	// SYS_ScanA: Is every 1s for one scan high
"SYS_ScanA_Tick1min"	M 5.6	BOOL	// SYS_ScanA: Is every min for one scan high
"SYS_ScanB_Tick200ms"	M 6.3	BOOL	// SYS_ScanB: Is every 200ms for one scan high
"SYS_ScanB_Tick500ms"	M 6.4	BOOL	// SYS_ScanB: Is every 500ms for one scan high
"SYS_ScanB_Tick1s"	M 6.5	BOOL	// SYS_ScanB: Is every 1s for one scan high
"SYS_ScanB_Tick1min"	M 6.6	BOOL	// SYS_ScanB: Is every min for one scan high
"SYS_ScanC_Tick200ms"	M 7.3	BOOL	// SYS_ScanC: Is every 200ms for one scan high
"SYS_ScanC_Tick500ms"	M 7.4	BOOL	// SYS_ScanC: Is every 500ms for one scan high
"SYS_ScanC_Tick1s"	M 7.5	BOOL	// SYS_ScanC: Is every 1s for one scan high
"SYS_ScanC_Tick1min"	M 7.6	BOOL	// SYS_ScanC: Is every min for one scan high
"SYS_infLog0"	M 9.0	BOOL	// SYS: Logical false all the time
"SYS_infLog1"	M 9.1	BOOL	// SYS: Logical true all the time
"SYS_CycleFlasher"	M 9.2	BOOL	// SYS: Status changing every scan
"SYS_Pulse500ms"	M 9.3	BOOL	// SYS: Pulse 500 ms true, 500ms false
"SYS_Pulse1000ms"	M 9.4	BOOL	// SYS: Pulse 1000ms true, 1000ms false
"SYS_Tick1s"	M 9.5	BOOL	// SYS: Tick is every 1s for one scan high
"GCS7_Gr_OutTick100ms"	M 10.2	BOOL	// GCS7: Group control module
"GCS7_Gr_OutTick200ms"	M 10.3	BOOL	// GCS7: Group control module
"GCS7_Gr_OutTick500ms"	M 10.4	BOOL	// GCS7: Group control module
"GCS7_Gr_OutTick1s"	M 10.5	BOOL	// GCS7: Group control module
"GCS7_Gr_OutTick1min"	M 10.6	BOOL	// GCS7: Group control module
"GCS7_Gr_OutRestartPLC"	M 11.0	BOOL	// GCS7: Group control module
"GCS7_Gr_SimDPtoImage"	M 11.1	BOOL	// GCS7: 1=Simulator uses process image GCS7:  0=Simulator uses DB16/17
"GCS7_Gr_OutLogOff"	M 11.2	BOOL	// GCS7: Group control module
"GCS7_Gr_OutCallFast1"	M 11.4	BOOL	// GCS7: Group control module
"GCS7_Gr_OutCallFast2"	M 11.5	BOOL	// GCS7: Group control module
"GCS7_Gr_OutCallFast3"	M 11.6	BOOL	// GCS7: Group control module
"GCS7_Gr_InBrakeMill"	M 12.0	BOOL	// GCS7: Is set by DFCA, when any machine is stoppinf with brake
"GCS7_Gr_OutNext"	M 12.2	BOOL	// GCS7: Group control module
"GCS7_Gr_OutFaultReset"	M 12.3	BOOL	// GCS7: Group control module
"GCS7_Gr_OutManualOff"	M 12.4	BOOL	// GCS7: Group control module
"GCS7_Gr_OutManualOn"	M 12.5	BOOL	// GCS7: Group control module
"GCS7_Gr_OutReportAll"	M 12.6	BOOL	// GCS7: Group control module
"GCS7_Gr_InCBit1"	M 13.0	BOOL	// GCS7: Group control module
"GCS7_Gr_InCBit2"	M 13.1	BOOL	// GCS7: Group control module
"GCS7_Gr_InCBit3"	M 13.2	BOOL	// GCS7: Group control module
"GCS7_Gr_InCBit4"	M 13.3	BOOL	// GCS7: Group control module
"GCS7_Gr_InFault"	M 13.4	BOOL	// GCS7: Group control module
"GCS7_Gr_InManual"	M 13.5	BOOL	// GCS7: Group control module
"GCS7_Gr_InHeavyStartup"	M 13.6	BOOL	// GCS7: Group control module
"GCS7_Gr_InFaultFlag"	M 13.7	BOOL	// GCS7: Group control module
"GCS7_Gr_InHWStop"	M 15.0	BOOL	// GCS7: Group control module
"GCS7_Gr_InDPFault"	M 15.1	BOOL	// GCS7: Group control module
"GCS7_Gr_InForce"	M 15.3	BOOL	// GCS7: Group control module
"GCS7_Gr_InMaintWarning"	M 15.4	BOOL	// GCS7: Group control module - Any maintenance element has a warning
"GCS7_Gr_InMaintFault"	M 15.5	BOOL	// GCS7: Group control module - Any maintenance element has a fault
"ENG_RemarkFlag"	M 50.0	BOOL	// ENG: Remark to remove all that flags
"CPU_TimeFlagsCopy"	MB 1	BYTE	// CPU: System timing
"CPU_TimeFlags"	MB 2	BYTE	// CPU: System timing
"SYS_CyclePartioning"	MB 3	BYTE	// SYS: Cycle partitioning
"SYS_Scan0_Time"	MB 4	BYTE	// SYS_Scan0: Timer flag
"SYS_ScanA_Time"	MB 5	BYTE	// SYS_ScanA: Timer flag
"SYS_ScanB_Time"	MB 6	BYTE	// SYS_ScanB: Timer flag
"SYS_ScanC_Time"	MB 7	BYTE	// SYS_ScanC: Timer flag
"SYS_GeneralFlags"	MB 9	BYTE	// SYS: General flags
"GCS7_Gr_Tick"	MB 10	BYTE	// GCS7: Group control module
"GCS7_Gr_MainToElMa"	MB 11	BYTE	// GCS7: Information main prog. to element and machine
"GCS7_Gr_ElMaToGroup1"	MB 12	BYTE	// GCS7: Information Element and machine to group
"GCS7_Gr_ElMaToGroup2"	MB 13	BYTE	// GCS7: Information Element and machine to group
"GCS7_Gr_OutLine"	MB 14	BYTE	// GCS7: Group control module
"ENG_Settings"	MB 50	BYTE	// ENG: Engineering settings
"Gr_ParHornCode"	MW 16	WORD
"SYS_MainProgram"	OB 1	OB 1	// SYS: Main program
"SYS_TOD_INT1"	OB 10	OB 10	// SYS: Time of Day Interrupt 1
"SYS_TOD_INT2"	OB 11	OB 11	// SYS: Time of Day Interrupt 2
"SYS_DEL_INT1"	OB 20	OB 20	// SYS: Time Delay Interrupt 1
"SYS_DEL_INT2"	OB 21	OB 21	// SYS: Time Delay Interrupt 2
"SYS_CycInt5s"	OB 30	OB 30	// SYS: Cyclic interrupt 5 sec
"SYS_CycInt2s"	OB 31	OB 31	// SYS: Cyclic interrupt 2 sec
"SYS_CycInt500ms"	OB 33	OB 33	// SYS: Cyclic interrupt 500 ms
"SYS_CycInt200ms"	OB 34	OB 34	// SYS: Cyclic interrupt 200 ms
"SYS_CycInt20ms"	OB 35	OB 35	// SYS: Cyclic interrupt 20 ms
"SYS_CycInt50ms"	OB 36	OB 36	// SYS: Cyclic interrupt 50 ms
"SYS_CycInt100ms"	OB 37	OB 37	// SYS: Cyclic interrupt 100 ms
"SYS_CycInt10ms"	OB 38	OB 38	// SYS: Cyclic interrupt 10 ms
"SYS_HW_INT1"	OB 40	OB 40	// SYS: Hardware Interrupt 1
"SYS_HW_INT2"	OB 41	OB 41	// SYS: Hardware Interrupt 2
"SYS_CYCL_FLT"	OB 80	OB 80	// SYS: Cycle time fault
"SYS_PS_FLT"	OB 81	OB 81	// SYS: Power Supply Fault
"SYS_IO_FLT1"	OB 82	OB 82	// SYS: I/O Point Fault 1
"SYS_IO_FLT2"	OB 83	OB 83	// SYS: I/O Point Fault 2
"SYS_HW_CPUFault"	OB 84	OB 84	// HW: CPU hardware failure
"SYS_OBNL_FLT"	OB 85	OB 85	// SYS: OB Not Loaded Fault
"SYS_RACK_FLT"	OB 86	OB 86	// SYS: Loss of Rack Fault
"SYS_ComFailure"	OB 87	OB 87	// SYS: Communication Fault
"PLC_StUpNewstart"	OB 100	OB 100	// PLC: Startup program on newstart
"PLC_StUpRestart"	OB 101	OB 101	// PLC: Startup program on restart
"PLC_StUpColdstart"	OB 102	OB 102	// PLC: Startup program on coldstart
"SYS_PROG_ERR"	OB 121	OB 121	// SYS: Programming Error
"SYS_MOD_ERR"	OB 122	OB 122	// SYS: Module Access Error
"A_2591_BTE01_AI1"	PIW 568	WORD	// AIR TEMPERATURE BELOW FLOOR
"A_2591_BTE02_AI1"	PIW 570	WORD	// AIR TEMPERATURE ABOVE FLOOR
"A_2545_QXV21_AI1"	PIW 572	WORD	// REGULATING VALVE ACTUEL VALUE
"A_2545_QXV31_AI1"	PIW 574	WORD	// REGULATING VALVE ACTUEL VALUE
"A_2550_BEE01_AI1"	PIW 576	WORD	// EXHAUST FLAP ACTUEL VALUE
"A_2511_BZS49_AI1"	PIW 580	WORD	// TRAVELING DRIVE POSITION CHANNEL 1/2
"A_2551_BEE01_AI1"	PIW 592	WORD	//  FRESH FLAP ACTUEL VALUE
"A_2552_BEE01_AI1"	PIW 594	WORD	//  FRESH FLAP ACTUEL VALUE
"A_2591_BTE03_AI1"	PIW 596	WORD	// AIR TEMPERATURE BELOW FLOOR
"A_2591_BTE04_AI1"	PIW 598	WORD	// AIR TEMPERATURE ABOVE FLOOR
"A_2691_BTE01_AI1"	PIW 668	WORD	// AIR TEMPERATURE BELOW FLOOR
"A_2691_BTE02_AI1"	PIW 670	WORD	// AIR TEMPERATURE ABOVE FLOOR
"A_2645_QXV21_AI1"	PIW 672	WORD	// REGULATING VALVE ACTUEL VALUE
"A_2645_QXV31_AI1"	PIW 674	WORD	// REGULATING VALVE ACTUEL VALUE
"A_2650_BEE01_AI1"	PIW 676	WORD	// EXHAUST FLAP ACTUEL VALUE
"A_2611_BZS49_AI1"	PIW 680	WORD	// TRAVELING DRIVE POSITION CHANNEL 1/2
"A_2651_BEE01_AI1"	PIW 692	WORD	//  FRESH FLAP ACTUEL VALUE
"A_2652_BEE01_AI1"	PIW 694	WORD	//  FRESH FLAP ACTUEL VALUE
"A_2691_BTE03_AI1"	PIW 696	WORD	// AIR TEMPERATURE BELOW FLOOR
"A_2691_BTE04_AI1"	PIW 698	WORD	// AIR TEMPERATURE ABOVE FLOOR
"A_2791_BTE01_AI1"	PIW 768	WORD	// AIR TEMPERATURE BELOW FLOOR
"A_2791_BTE02_AI1"	PIW 770	WORD	// AIR TEMPERATURE ABOVE FLOOR
"A_2745_QXV21_AI1"	PIW 772	WORD	// REGULATING VALVE ACTUEL VALUE
"A_2745_QXV31_AI1"	PIW 774	WORD	// REGULATING VALVE ACTUEL VALUE
"A_2750_BEE01_AI1"	PIW 776	WORD	// EXHAUST FLAP ACTUEL VALUE
"A_2711_BZS49_AI1"	PIW 780	WORD	// TRAVELING DRIVE POSITION CHANNEL 1/2
"A_2751_BEE01_AI1"	PIW 792	WORD	//  FRESH FLAP ACTUEL VALUE
"A_2752_BEE01_AI1"	PIW 794	WORD	//  FRESH FLAP ACTUEL VALUE
"A_2791_BTE03_AI1"	PIW 796	WORD	// AIR TEMPERATURE BELOW FLOOR
"A_2791_BTE04_AI1"	PIW 798	WORD	// AIR TEMPERATURE ABOVE FLOOR
"A_2891_BTE01_AI1"	PIW 868	WORD	// AIR TEMPERATURE BELOW FLOOR
"A_2891_BTE02_AI1"	PIW 870	WORD	// AIR TEMPERATURE ABOVE FLOOR
"A_2845_QXV21_AI1"	PIW 872	WORD	// REGULATING VALVE ACTUEL VALUE
"A_2845_QXV31_AI1"	PIW 874	WORD	// REGULATING VALVE ACTUEL VALUE
"A_2850_BEE01_AI1"	PIW 876	WORD	// EXHAUST FLAP ACTUEL VALUE
"A_2811_BZS49_AI1"	PIW 880	WORD	// TRAVELING DRIVE POSITION CHANNEL 1/2
"A_2851_BEE01_AI1"	PIW 892	WORD	//  FRESH FLAP ACTUEL VALUE
"A_2852_BEE01_AI1"	PIW 894	WORD	//  FRESH FLAP ACTUEL VALUE
"A_2891_BTE03_AI1"	PIW 896	WORD	// AIR TEMPERATURE BELOW FLOOR
"A_2891_BTE04_AI1"	PIW 898	WORD	// AIR TEMPERATURE ABOVE FLOOR
"A_3125_BTE05_AI1"	PIW 928	WORD	// TEMPERATURE BEARING TEMPERATUR SENSOR
"A_3125_BTE06_AI1"	PIW 930	WORD	// TEMPERATURE BEARING TEMPERATUR SENSOR
"A_3126_BTE05_AI1"	PIW 932	WORD	// TEMPERATURE BEARING TEMPERATUR SENSOR
"A_3126_BTE06_AI1"	PIW 934	WORD	// TEMPERATURE BEARING TEMPERATUR SENSOR
"A_3191_BTE01_AI1"	PIW 936	WORD	// AIR TEMPERATURE BELOW FLOOR
"A_3191_BTE05_AI1"	PIW 938	WORD	// AIR TEMPERATURE DIFFUSOR FAN 1
"A_3191_BTE07_AI1"	PIW 940	WORD	// AIR TEMPERATURE ABOVE FLOOR
"A_3191_BTE08_AI1"	PIW 942	WORD	// AIR TEMPERATURE AFTER BURNER 1
"A_3191_BTE10_AI1"	PIW 944	WORD	// AIR TEMPERATURE BEFORE BURNER 2
"A_3191_BTE11_AI1"	PIW 946	WORD	// AIR TEMPERATURE AMBIENT AIR
"A_3191_BTE12_AI1"	PIW 948	WORD	// AIR TEMPERATURE AFTER HEAT EXCHANGER FLAP
"A_3191_BTE06_AI1"	PIW 950	WORD	// AIR TEMPERATURE DIFFUSOR FAN 2
"A_3125_KCU04_AI2"	PIW 952	WORD	// VIBRATION MONITOR FAN 1 CHANNEL 2
"A_3125_KCU04_AI1"	PIW 954	WORD	// VIBRATION MONITOR FAN 1 CHANNEL 1
"A_3126_KCU04_AI2"	PIW 956	WORD	// VIBRATION MONITOR FAN 2 CHANNEL 2
"A_3126_KCU04_AI1"	PIW 958	WORD	// VIBRATION MONITOR FAN 2 CHANNEL 1
"A_3161_KCL11_AI1"	PIW 960	WORD	// BURNER 1 INPUT SIGNAL ANALOG
"A_3161_KCL12_AI1"	PIW 962	WORD	// BURNER 2 INPUT SIGNAL ANALOG
"A_3111_BZS24_AI1"	PIW 964	WORD	// LIFTING DRIVE POSITION CHANNEL 1/2
"A_3111_BZS34_AI1"	PIW 976	WORD	// LIFTING DRIVE POSITION CHANNEL 1/2
"A_3121_BZS46_AI1"	PIW 988	WORD	// TRAVELING DRIVE POSITION CHANNEL 1/2
"A_3225_BTE05_AI1"	PIW 1028	WORD	// TEMPERATURE BEARING TEMPERATUR SENSOR
"A_3225_BTE06_AI1"	PIW 1030	WORD	// TEMPERATURE BEARING TEMPERATUR SENSOR
"A_3226_BTE05_AI1"	PIW 1032	WORD	// TEMPERATURE BEARING TEMPERATUR SENSOR
"A_3226_BTE06_AI1"	PIW 1034	WORD	// TEMPERATURE BEARING TEMPERATUR SENSOR
"A_3291_BTE01_AI1"	PIW 1036	WORD	// AIR TEMPERATURE BELOW FLOOR
"A_3291_BTE05_AI1"	PIW 1038	WORD	// AIR TEMPERATURE DIFFUSOR FAN 1
"A_3291_BTE07_AI1"	PIW 1040	WORD	// AIR TEMPERATURE ABOVE FLOOR
"A_3291_BTE08_AI1"	PIW 1042	WORD	// AIR TEMPERATURE AFTER BURNER 1
"A_3291_BTE10_AI1"	PIW 1044	WORD	// AIR TEMPERATURE BEFORE BURNER 3
"A_3291_BTE14_AI1"	PIW 1048	WORD	// AIR TEMPERATURE ON THE MIDDLE KILN2
"A_3291_BTE06_AI1"	PIW 1050	WORD	// AIR TEMPERATURE DIFFUSOR FAN 2
"A_3225_KCU04_AI2"	PIW 1052	WORD	// VIBRATION MONITOR FAN 1 CHANNEL 2
"A_3225_KCU04_AI1"	PIW 1054	WORD	// VIBRATION MONITOR FAN 1 CHANNEL 1
"A_3226_KCU04_AI2"	PIW 1056	WORD	// VIBRATION MONITOR FAN 2 CHANNEL 2
"A_3226_KCU04_AI1"	PIW 1058	WORD	// VIBRATION MONITOR FAN 2 CHANNEL 1
"A_3261_KCL11_AI1"	PIW 1060	WORD	// BURNER 3 INPUT SIGNAL ANALOG
"A_3211_BZS24_AI1"	PIW 1064	WORD	// LIFTING DRIVE POSITION CHANNEL 1/2
"A_3211_BZS34_AI1"	PIW 1076	WORD	// LIFTING DRIVE POSITION CHANNEL 1/2
"A_3221_BZS46_AI1"	PIW 1088	WORD	// TRAVELING DRIVE POSITION CHANNEL 1/2
"A_3930_PII24_O1"	PIW 1160	WORD	// CURRENT MEASURING
"A_3945_PII24_O1"	PIW 1162	WORD	// CURRENT MEASURING
"A_6105_PII35_AI1"	PIW 1200	WORD	// ACT. CURRENT ELEVATOR 6105
"A_6163_PII35_AI1"	PIW 1202	WORD	// ACT. CURRENT ELEVATOR 6163
"A_2545_QXV21_AO1"	PQW 568	WORD	// REGULATING VALVE SET POINT
"A_2545_QXV31_AO1"	PQW 570	WORD	// REGULATING VALVE SET POINT
"A_2645_QXV21_AO1"	PQW 668	WORD	// REGULATING VALVE SET POINT
"A_2645_QXV31_AO1"	PQW 670	WORD	// REGULATING VALVE SET POINT
"A_2745_QXV21_AO1"	PQW 768	WORD	// REGULATING VALVE SET POINT
"A_2745_QXV31_AO1"	PQW 770	WORD	// REGULATING VALVE SET POINT
"A_2845_QXV21_AO1"	PQW 868	WORD	// REGULATING VALVE SET POINT
"A_2845_QXV31_AO1"	PQW 870	WORD	// REGULATING VALVE SET POINT
"A_3161_KCL11_AO1"	PQW 928	WORD	// BURNER 1 OUTPUT SIGNAL ANALOG
"A_3161_KCL12_AO1"	PQW 930	WORD	// BURNER 2 OUTPUT SIGNAL ANALOG
"A_3261_KCL11_AO1"	PQW 1028	WORD	// BURNER 3 OUTPUT SIGNAL ANALOG
"A_1199_PAZ11_O1"	Q 16.0	BOOL	// ALARM HORN
"A_1111_MXZ11_O1"	Q 24.0	BOOL	// ASPIRATION FAN TANK 1
"A_1112_MXZ11_O1"	Q 24.1	BOOL	// ASPIRATION FAN TANK 2
